C07189=1028.649,297.981,-127.130,170.913,46.438,158.974
C07190=1028.655,298.229,-127.163,170.917,46.437,158.975
C07191=1028.663,298.477,-127.195,170.922,46.437,158.975
C07192=1028.669,298.724,-127.228,170.927,46.436,158.976
C07193=1028.676,298.972,-127.261,170.931,46.436,158.976
C07194=1028.683,299.220,-127.293,170.935,46.436,158.976
C07195=1028.689,299.468,-127.326,170.941,46.435,158.977
C07196=1028.696,299.716,-127.359,170.945,46.435,158.977
C07197=1028.703,299.963,-127.391,170.949,46.434,158.978
C07198=1028.710,300.211,-127.424,170.954,46.434,158.978
C07199=1028.717,300.459,-127.457,170.959,46.432,158.978
C07200=1028.724,300.706,-127.490,170.963,46.432,158.979
C07201=1028.731,300.954,-127.523,170.967,46.432,158.979
C07202=1028.737,301.202,-127.556,170.972,46.431,158.980
C07203=1028.744,301.449,-127.588,170.977,46.431,158.980
C07204=1028.751,301.697,-127.621,170.981,46.430,158.981
C07205=1028.757,301.945,-127.654,170.986,46.430,158.981
C07206=1028.765,302.192,-127.687,170.991,46.429,158.981
C07207=1028.772,302.440,-127.720,170.995,46.429,158.982
C07208=1028.778,302.688,-127.753,171.000,46.428,158.982
C07209=1028.785,302.936,-127.786,171.005,46.428,158.983
C07210=1028.793,303.183,-127.819,171.010,46.428,158.983
C07211=1028.799,303.431,-127.852,171.014,46.427,158.984
C07212=1028.806,303.679,-127.885,171.019,46.427,158.984
C07213=1028.813,303.926,-127.917,171.024,46.426,158.985
C07214=1028.820,304.174,-127.951,171.028,46.426,158.985
C07215=1028.826,304.421,-127.984,171.033,46.425,158.986
C07216=1028.834,304.669,-128.017,171.038,46.425,158.986
C07217=1028.841,304.917,-128.050,171.042,46.424,158.986
C07218=1028.847,305.165,-128.083,171.047,46.424,158.987
C07219=1028.855,305.412,-128.117,171.052,46.423,158.987
C07220=1028.862,305.660,-128.149,171.056,46.424,158.988
C07221=1028.869,305.907,-128.183,171.062,46.423,158.988
C07222=1028.880,306.326,-128.238,171.069,46.422,158.989
C07223=1028.893,306.744,-128.294,171.077,46.422,158.990
C07224=1028.904,307.163,-128.350,171.086,46.421,158.991
C07225=1028.916,307.582,-128.406,171.093,46.420,158.992
C07226=1028.923,307.828,-128.439,171.099,46.420,158.992
C07227=1028.931,308.076,-128.473,171.103,46.419,158.992
C07228=1028.937,308.324,-128.506,171.107,46.419,158.993
C07229=1028.945,308.572,-128.539,171.113,46.419,158.994
C07230=1028.952,308.819,-128.572,171.117,46.418,158.994
C07231=1028.959,309.067,-128.606,171.122,46.418,158.994
C07232=1028.966,309.315,-128.640,171.127,46.418,158.995
C07233=1028.974,309.563,-128.672,171.132,46.417,158.996
C07234=1028.980,309.810,-128.706,171.137,46.417,158.996
C07235=1028.988,310.057,-128.740,171.141,46.417,158.997
C07236=1028.995,310.305,-128.773,171.147,46.416,158.997
C07237=1029.002,310.553,-128.806,171.151,46.416,158.997
C07238=1029.009,310.800,-128.839,171.157,46.416,158.998
C07239=1029.016,311.048,-128.873,171.161,46.415,158.998
C07240=1029.023,311.295,-128.907,171.167,46.415,158.999
C07241=1029.031,311.543,-128.941,171.171,46.415,159.000
C07242=1029.036,311.790,-128.975,171.176,46.415,159.000
C07243=1029.044,312.038,-129.009,171.181,46.415,159.001
C07244=1029.051,312.286,-129.043,171.185,46.415,159.001
C07245=1029.057,312.534,-129.077,171.190,46.415,159.002
C07246=1029.064,312.780,-129.110,171.196,46.415,159.002
C07247=1029.071,313.028,-129.144,171.200,46.415,159.003
C07248=1029.078,313.276,-129.179,171.206,46.414,159.004
C07249=1029.085,313.523,-129.213,171.210,46.415,159.004
C07250=1029.091,313.770,-129.247,171.215,46.414,159.005
C07251=1029.098,314.018,-129.281,171.220,46.414,159.005
C07252=1029.105,314.266,-129.315,171.225,46.414,159.006
C07253=1029.112,314.514,-129.349,171.230,46.414,159.006
C07254=1029.119,314.761,-129.384,171.235,46.414,159.007
C07255=1029.126,315.009,-129.418,171.240,46.414,159.008
C07256=1029.132,315.256,-129.452,171.245,46.414,159.008
C07257=1029.140,315.503,-129.486,171.251,46.414,159.009
C07258=1029.147,315.751,-129.520,171.255,46.414,159.009
C07259=1029.153,315.999,-129.555,171.260,46.414,159.010
C07260=1029.161,316.246,-129.588,171.265,46.414,159.010
C07261=1029.168,316.493,-129.623,171.270,46.414,159.011
C07262=1029.175,316.741,-129.657,171.275,46.414,159.012
C07263=1029.182,316.989,-129.691,171.280,46.414,159.012
C07264=1029.189,317.236,-129.726,171.286,46.414,159.013
C07265=1029.196,317.484,-129.760,171.290,46.414,159.013
C07266=1029.203,317.732,-129.794,171.296,46.414,159.014
C07267=1029.210,317.979,-129.829,171.300,46.414,159.015
C07268=1029.217,318.227,-129.863,171.306,46.414,159.015
C07269=1029.225,318.474,-129.897,171.311,46.414,159.016
C07270=1029.231,318.722,-129.932,171.316,46.414,159.016
C07271=1029.238,318.969,-129.966,171.321,46.414,159.017
C07272=1029.245,319.217,-130.001,171.326,46.414,159.018
C07273=1029.252,319.464,-130.035,171.331,46.414,159.018
C07274=1029.260,319.711,-130.069,171.337,46.414,159.019
C07275=1029.266,319.959,-130.104,171.341,46.414,159.020
C07276=1029.274,320.206,-130.139,171.347,46.414,159.020
C07277=1029.281,320.454,-130.173,171.351,46.415,159.021
C07278=1029.287,320.665,-130.202,171.356,46.415,159.021
C07279=1029.293,320.878,-130.232,171.360,46.414,159.022
C07280=1029.300,321.089,-130.262,171.365,46.415,159.022
C07281=1029.306,321.301,-130.291,171.370,46.415,159.023
C07282=1029.311,321.512,-130.321,171.374,46.415,159.024
C07283=1029.317,321.724,-130.350,171.379,46.415,159.024
C07284=1029.324,321.936,-130.381,171.383,46.415,159.025
C07285=1029.330,322.147,-130.410,171.388,46.415,159.025
C07286=1029.337,322.395,-130.445,171.392,46.415,159.026
C07287=1029.345,322.642,-130.479,171.398,46.415,159.026
C07288=1029.351,322.890,-130.514,171.403,46.416,159.027
C07289=1029.360,323.137,-130.549,171.409,46.416,159.028
C07290=1029.366,323.385,-130.584,171.414,46.416,159.028
C07291=1029.374,323.632,-130.618,171.419,46.416,159.029
C07292=1029.381,323.879,-130.652,171.424,46.416,159.030
C07293=1029.388,324.127,-130.688,171.429,46.416,159.030
C07294=1029.396,324.375,-130.722,171.435,46.417,159.031
C07295=1029.403,324.622,-130.757,171.441,46.417,159.032
C07296=1029.410,324.869,-130.792,171.445,46.417,159.032
C07297=1029.418,325.117,-130.827,171.451,46.417,159.033
C07298=1029.425,325.364,-130.862,171.457,46.417,159.034
C07299=1029.433,325.611,-130.896,171.461,46.417,159.034
C07300=1029.440,325.859,-130.932,171.467,46.417,159.035
C07301=1029.447,326.106,-130.966,171.473,46.418,159.036
C07302=1029.455,326.354,-131.002,171.478,46.418,159.037
C07303=1029.462,326.601,-131.036,171.483,46.418,159.037
C07304=1029.470,326.848,-131.071,171.489,46.419,159.038
C07305=1029.477,327.096,-131.106,171.494,46.419,159.039
C07306=1029.485,327.344,-131.141,171.499,46.419,159.039
C07307=1029.492,327.592,-131.177,171.505,46.419,159.040
C07308=1029.500,327.839,-131.211,171.510,46.420,159.041
C07309=1029.506,328.086,-131.246,171.516,46.420,159.042
C07310=1029.514,328.333,-131.282,171.521,46.420,159.042
C07311=1029.521,328.581,-131.318,171.526,46.421,159.043
C07312=1029.528,328.828,-131.353,171.532,46.421,159.044
C07313=1029.535,329.076,-131.389,171.538,46.421,159.044
C07314=1029.543,329.323,-131.423,171.543,46.422,159.045
C07315=1029.550,329.571,-131.459,171.548,46.422,159.046
C07316=1029.557,329.817,-131.495,171.554,46.423,159.047
C07317=1029.565,330.066,-131.530,171.559,46.423,159.047
C07318=1029.572,330.312,-131.566,171.565,46.423,159.048
C07319=1029.578,330.560,-131.601,171.571,46.424,159.049
C07320=1029.586,330.807,-131.638,171.576,46.425,159.050
C07321=1029.594,331.054,-131.672,171.581,46.425,159.050
C07322=1029.601,331.302,-131.708,171.587,46.425,159.051
C07323=1029.608,331.549,-131.743,171.593,46.426,159.052
C07324=1029.616,331.796,-131.780,171.598,46.427,159.053
C07325=1029.623,332.045,-131.815,171.604,46.426,159.053
C07326=1029.630,332.291,-131.851,171.610,46.427,159.054
C07327=1029.638,332.539,-131.887,171.615,46.428,159.055
C07328=1029.645,332.786,-131.922,171.620,46.428,159.056
C07329=1029.653,333.033,-131.958,171.626,46.429,159.057
C07330=1029.660,333.280,-131.994,171.632,46.429,159.058
C07331=1029.667,333.528,-132.029,171.638,46.429,159.058
C07332=1029.675,333.775,-132.066,171.643,46.430,159.059
C07333=1029.682,334.022,-132.101,171.649,46.431,159.060
C07334=1029.690,334.270,-132.137,171.655,46.431,159.061
C07335=1029.697,334.518,-132.173,171.660,46.432,159.061
C07336=1029.704,334.764,-132.209,171.665,46.433,159.062
C07337=1029.712,335.012,-132.245,171.671,46.433,159.063
C07338=1029.718,335.222,-132.276,171.676,46.434,159.064
C07339=1029.724,335.431,-132.307,171.681,46.434,159.064
C07340=1029.730,335.641,-132.337,171.686,46.435,159.065
C07341=1029.737,335.849,-132.368,171.690,46.435,159.066
C07342=1029.743,336.059,-132.398,171.695,46.436,159.067
C07343=1029.749,336.269,-132.429,171.700,46.437,159.067
C07344=1029.756,336.478,-132.459,171.706,46.437,159.068
C07345=1029.762,336.687,-132.490,171.711,46.437,159.069
C07346=1029.769,336.935,-132.526,171.716,46.438,159.069
C07347=1029.776,337.182,-132.562,171.721,46.439,159.070
C07348=1029.784,337.429,-132.600,171.727,46.439,159.071
C07349=1029.791,337.676,-132.636,171.734,46.440,159.072
C07350=1029.799,337.924,-132.672,171.740,46.441,159.073
C07351=1029.807,338.171,-132.708,171.745,46.441,159.074
C07352=1029.814,338.418,-132.744,171.750,46.442,159.075
C07353=1029.821,338.665,-132.780,171.756,46.443,159.075
C07354=1029.829,338.913,-132.816,171.762,46.444,159.076
C07355=1029.837,339.160,-132.853,171.768,46.444,159.077
C07356=1029.844,339.407,-132.890,171.774,46.445,159.078
C07357=1029.851,339.654,-132.926,171.781,46.446,159.079
C07358=1029.859,339.901,-132.962,171.786,46.447,159.080
C07359=1029.867,340.148,-132.999,171.791,46.447,159.081
C07360=1029.874,340.396,-133.035,171.798,46.449,159.082
C07361=1029.881,340.643,-133.072,171.803,46.449,159.083
C07362=1029.889,340.890,-133.109,171.809,46.450,159.083
C07363=1029.897,341.138,-133.145,171.816,46.451,159.084
C07364=1029.904,341.385,-133.183,171.822,46.451,159.085
C07365=1029.912,341.632,-133.219,171.828,46.452,159.086
C07366=1029.919,341.878,-133.256,171.834,46.453,159.087
C07367=1029.926,342.126,-133.293,171.840,46.454,159.088
C07368=1029.934,342.373,-133.329,171.846,46.455,159.089
C07369=1029.941,342.621,-133.366,171.851,46.456,159.090
C07370=1029.949,342.868,-133.403,171.857,46.457,159.091
C07371=1029.957,343.114,-133.440,171.863,46.458,159.092
C07372=1029.964,343.362,-133.477,171.869,46.459,159.093
C07373=1029.972,343.609,-133.514,171.875,46.459,159.094
C07374=1029.979,343.856,-133.551,171.881,46.461,159.095
C07375=1029.987,344.104,-133.588,171.888,46.462,159.096
C07376=1029.995,344.350,-133.625,171.894,46.462,159.096
C07377=1030.002,344.598,-133.662,171.900,46.463,159.097
C07378=1030.010,344.844,-133.699,171.906,46.464,159.098
C07379=1030.017,345.092,-133.736,171.912,46.466,159.099
C07380=1030.026,345.340,-133.773,171.918,46.466,159.100
C07381=1030.033,345.587,-133.811,171.924,46.467,159.101
C07382=1030.041,345.834,-133.848,171.931,46.468,159.102
C07383=1030.048,346.081,-133.885,171.937,46.469,159.103
C07384=1030.056,346.328,-133.922,171.943,46.471,159.104
C07385=1030.063,346.575,-133.960,171.949,46.471,159.105
C07386=1030.071,346.822,-133.996,171.955,46.472,159.106
C07387=1030.079,347.069,-134.034,171.961,46.473,159.107
C07388=1030.087,347.316,-134.071,171.968,46.474,159.108
C07389=1030.094,347.563,-134.109,171.974,46.476,159.109
C07390=1030.102,347.810,-134.146,171.980,46.477,159.110
C07391=1030.110,348.057,-134.183,171.986,46.478,159.111
C07392=1030.118,348.304,-134.220,171.992,46.479,159.112
C07393=1030.125,348.552,-134.258,171.999,46.480,159.113
C07394=1030.133,348.799,-134.296,172.005,46.481,159.114
C07395=1030.141,349.046,-134.333,172.011,46.482,159.115
C07396=1030.148,349.292,-134.371,172.017,46.483,159.116
C07397=1030.156,349.540,-134.409,172.024,46.484,159.117
C07398=1030.169,349.956,-134.471,172.035,46.486,159.119
C07399=1030.181,350.371,-134.535,172.046,46.488,159.121
C07400=1030.195,350.787,-134.599,172.056,46.490,159.123
C07401=1030.208,351.203,-134.662,172.067,46.492,159.124
C07402=1030.215,351.449,-134.700,172.073,46.494,159.126
C07403=1030.223,351.697,-134.738,172.080,46.495,159.127
C07404=1030.231,351.943,-134.776,172.086,46.496,159.128
C07405=1030.239,352.191,-134.813,172.092,46.497,159.129
C07406=1030.247,352.437,-134.852,172.099,46.499,159.130
C07407=1030.254,352.685,-134.889,172.106,46.500,159.131
C07408=1030.262,352.932,-134.928,172.112,46.501,159.132
C07409=1030.271,353.178,-134.965,172.119,46.503,159.133
C07410=1030.279,353.426,-135.003,172.125,46.504,159.134
C07411=1030.286,353.672,-135.042,172.131,46.506,159.135
C07412=1030.294,353.920,-135.080,172.139,46.506,159.136
C07413=1030.301,354.167,-135.118,172.145,46.508,159.138
C07414=1030.310,354.414,-135.156,172.151,46.509,159.139
C07415=1030.318,354.660,-135.194,172.157,46.510,159.140
C07416=1030.326,354.907,-135.233,172.164,46.512,159.141
C07417=1030.333,355.154,-135.270,172.172,46.514,159.142
C07418=1030.341,355.402,-135.309,172.178,46.515,159.143
C07419=1030.349,355.648,-135.347,172.184,46.516,159.144
C07420=1030.358,355.895,-135.385,172.190,46.517,159.145
C07421=1030.365,356.142,-135.423,172.198,46.519,159.146
C07422=1030.374,356.389,-135.462,172.204,46.521,159.148
C07423=1030.381,356.635,-135.500,172.211,46.522,159.149
C07424=1030.389,356.883,-135.539,172.217,46.523,159.150
C07425=1030.397,357.130,-135.577,172.225,46.525,159.151
C07426=1030.405,357.376,-135.616,172.231,46.527,159.152
C07427=1030.413,357.623,-135.654,172.237,46.528,159.153
C07428=1030.421,357.870,-135.692,172.244,46.529,159.155
C07429=1030.429,358.117,-135.731,172.252,46.531,159.156
C07430=1030.437,358.364,-135.770,172.258,46.532,159.157
C07431=1030.445,358.610,-135.809,172.265,46.534,159.158
C07432=1030.453,358.858,-135.847,172.272,46.536,159.159
C07433=1030.461,359.105,-135.886,172.278,46.537,159.160
C07434=1030.469,359.352,-135.924,172.285,46.538,159.162
C07435=1030.477,359.598,-135.963,172.292,46.540,159.163
C07436=1030.485,359.845,-136.002,172.299,46.542,159.164
C07437=1030.493,360.092,-136.041,172.305,46.543,159.165
C07438=1030.502,360.339,-136.080,172.313,46.545,159.167
C07439=1030.509,360.586,-136.119,172.319,46.546,159.168
C07440=1030.517,360.832,-136.158,172.326,46.548,159.169
C07441=1030.525,361.080,-136.197,172.333,46.549,159.170
C07442=1030.534,361.326,-136.236,172.340,46.552,159.172
C07443=1030.542,361.573,-136.275,172.347,46.553,159.173
C07444=1030.549,361.820,-136.314,172.354,46.555,159.174
C07445=1030.557,362.067,-136.353,172.361,46.557,159.175
C07446=1030.566,362.313,-136.392,172.369,46.559,159.177
C07447=1030.573,362.560,-136.432,172.375,46.560,159.178
C07448=1030.582,362.807,-136.471,172.382,46.562,159.179
C07449=1030.590,363.054,-136.510,172.389,46.563,159.180
C07450=1030.598,363.300,-136.549,172.396,46.566,159.182
C07451=1030.606,363.547,-136.589,172.404,46.567,159.183
C07452=1030.614,363.794,-136.627,172.410,46.569,159.184
C07453=1030.622,364.041,-136.667,172.418,46.571,159.186
C07454=1030.629,364.252,-136.701,172.423,46.572,159.187
C07455=1030.637,364.463,-136.735,172.430,46.574,159.188
C07456=1030.643,364.673,-136.768,172.436,46.575,159.189
C07457=1030.650,364.884,-136.802,172.441,46.577,159.190
C07458=1030.657,365.096,-136.836,172.448,46.578,159.191
C07459=1030.665,365.307,-136.869,172.454,46.580,159.192
C07460=1030.671,365.518,-136.903,172.460,46.582,159.194
C07461=1030.678,365.729,-136.937,172.466,46.583,159.195
C07462=1030.686,365.976,-136.976,172.474,46.585,159.196
C07463=1030.694,366.222,-137.016,172.480,46.587,159.197
C07464=1030.703,366.468,-137.056,172.488,46.589,159.199
C07465=1030.711,366.715,-137.096,172.495,46.591,159.200
C07466=1030.719,366.962,-137.135,172.503,46.592,159.201
C07467=1030.728,367.209,-137.175,172.509,46.595,159.203
C07468=1030.736,367.456,-137.215,172.517,46.597,159.204
C07469=1030.745,367.703,-137.254,172.525,46.598,159.205
C07470=1030.753,367.949,-137.293,172.532,46.600,159.207
C07471=1030.761,368.195,-137.334,172.539,46.602,159.208
C07472=1030.770,368.442,-137.373,172.546,46.605,159.210
C07473=1030.779,368.689,-137.413,172.554,46.606,159.211
C07474=1030.787,368.936,-137.454,172.562,46.608,159.212
C07475=1030.795,369.182,-137.493,172.569,46.610,159.214
C07476=1030.803,369.429,-137.533,172.576,46.612,159.215
C07477=1030.812,369.675,-137.573,172.583,46.615,159.217
C07478=1030.820,369.923,-137.613,172.591,46.617,159.218
C07479=1030.828,370.169,-137.654,172.599,46.619,159.219
C07480=1030.837,370.415,-137.694,172.606,46.621,159.221
C07481=1030.844,370.662,-137.734,172.613,46.623,159.222
C07482=1030.853,370.909,-137.775,172.621,46.625,159.224
C07483=1030.862,371.155,-137.815,172.628,46.627,159.225
C07484=1030.870,371.402,-137.855,172.636,46.629,159.227
C07485=1030.878,371.649,-137.896,172.644,46.632,159.228
C07486=1030.887,371.895,-137.936,172.651,46.634,159.230
C07487=1030.895,372.142,-137.976,172.659,46.636,159.231
C07488=1030.903,372.389,-138.017,172.667,46.638,159.232
C07489=1030.912,372.635,-138.057,172.674,46.640,159.234
C07490=1030.920,372.881,-138.097,172.682,46.643,159.235
C07491=1030.929,373.128,-138.138,172.689,46.645,159.237
C07492=1030.937,373.374,-138.178,172.697,46.646,159.238
C07493=1030.946,373.621,-138.219,172.705,46.649,159.240
C07494=1030.954,373.867,-138.260,172.712,46.651,159.241
C07495=1030.963,374.113,-138.300,172.720,46.653,159.243
C07496=1030.972,374.360,-138.341,172.728,46.656,159.244
C07497=1030.980,374.606,-138.382,172.736,46.658,159.246
C07498=1030.989,374.853,-138.422,172.743,46.661,159.248
C07499=1030.997,375.099,-138.463,172.751,46.663,159.249
C07500=1031.006,375.346,-138.504,172.759,46.665,159.251
C07501=1031.015,375.593,-138.544,172.767,46.667,159.252
C07502=1031.023,375.839,-138.585,172.775,46.670,159.254
C07503=1031.032,376.086,-138.627,172.783,46.672,159.255
C07504=1031.041,376.332,-138.667,172.791,46.674,159.257
C07505=1031.049,376.578,-138.708,172.798,46.677,159.258
C07506=1031.058,376.825,-138.749,172.806,46.679,159.260
C07507=1031.067,377.071,-138.789,172.814,46.681,159.261
C07508=1031.076,377.318,-138.830,172.822,46.684,159.263
C07509=1031.085,377.564,-138.872,172.830,46.686,159.265
C07510=1031.093,377.810,-138.913,172.838,46.688,159.266
C07511=1031.102,378.057,-138.954,172.846,46.691,159.268
C07512=1031.110,378.304,-138.995,172.855,46.694,159.269
C07513=1031.118,378.549,-139.037,172.863,46.696,159.271
C07514=1031.127,378.771,-139.074,172.870,46.698,159.272
C07515=1031.135,378.992,-139.111,172.877,46.701,159.274
C07516=1031.142,379.214,-139.148,172.885,46.703,159.276
C07517=1031.150,379.436,-139.185,172.891,46.705,159.277
C07518=1031.158,379.657,-139.222,172.899,46.708,159.279
C07519=1031.165,379.879,-139.260,172.906,46.710,159.280
C07520=1031.173,380.100,-139.297,172.913,46.712,159.281
C07521=1031.181,380.322,-139.334,172.921,46.715,159.283
C07522=1031.190,380.568,-139.376,172.930,46.717,159.285
C07523=1031.199,380.814,-139.417,172.938,46.720,159.286
C07524=1031.207,381.060,-139.459,172.946,46.722,159.288
C07525=1031.216,381.307,-139.501,172.954,46.725,159.290
C07526=1031.225,381.553,-139.543,172.962,46.728,159.291
C07527=1031.234,381.799,-139.585,172.971,46.730,159.293
C07528=1031.242,382.046,-139.626,172.979,46.733,159.295
C07529=1031.251,382.292,-139.668,172.987,46.736,159.297
C07530=1031.260,382.539,-139.710,172.995,46.739,159.298
C07531=1031.269,382.785,-139.751,173.004,46.741,159.300
C07532=1031.278,383.031,-139.793,173.012,46.744,159.302
C07533=1031.287,383.277,-139.836,173.020,46.747,159.303
C07534=1031.296,383.523,-139.877,173.030,46.750,159.305
C07535=1031.305,383.770,-139.919,173.038,46.752,159.307
C07536=1031.314,384.016,-139.961,173.046,46.755,159.309
C07537=1031.323,384.262,-140.003,173.054,46.758,159.310
C07538=1031.332,384.508,-140.045,173.063,46.761,159.312
C07539=1031.341,384.755,-140.087,173.072,46.764,159.314
C07540=1031.351,385.000,-140.129,173.080,46.766,159.316
C07541=1031.360,385.247,-140.171,173.089,46.769,159.318
C07542=1031.369,385.493,-140.214,173.097,46.772,159.319
C07543=1031.378,385.740,-140.255,173.106,46.775,159.321
C07544=1031.387,385.986,-140.297,173.115,46.778,159.323
C07545=1031.396,386.232,-140.339,173.124,46.781,159.325
C07546=1031.406,386.477,-140.382,173.132,46.784,159.327
C07547=1031.415,386.725,-140.425,173.141,46.786,159.328
C07548=1031.424,386.970,-140.467,173.150,46.789,159.330
C07549=1031.433,387.217,-140.509,173.158,46.792,159.332
C07550=1031.442,387.463,-140.551,173.167,46.795,159.334
C07551=1031.451,387.709,-140.595,173.176,46.798,159.336
C07552=1031.460,387.955,-140.637,173.184,46.801,159.338
C07553=1031.470,388.201,-140.679,173.193,46.804,159.339
C07554=1031.479,388.448,-140.723,173.203,46.807,159.341
C07555=1031.488,388.693,-140.765,173.211,46.810,159.343
C07556=1031.497,388.939,-140.808,173.220,46.814,159.345
C07557=1031.507,389.186,-140.850,173.229,46.816,159.347
C07558=1031.515,389.432,-140.893,173.238,46.819,159.349
C07559=1031.525,389.677,-140.936,173.247,46.823,159.351
C07560=1031.535,389.924,-140.979,173.256,46.826,159.353
C07561=1031.543,390.170,-141.022,173.265,46.829,159.355
C07562=1031.553,390.416,-141.065,173.274,46.832,159.357
C07563=1031.561,390.662,-141.108,173.283,46.835,159.359
C07564=1031.571,390.908,-141.151,173.292,46.838,159.360
C07565=1031.580,391.154,-141.194,173.301,46.842,159.363
C07566=1031.589,391.400,-141.237,173.310,46.844,159.364
C07567=1031.599,391.646,-141.281,173.319,46.848,159.366
C07568=1031.608,391.892,-141.323,173.329,46.851,159.369
C07569=1031.617,392.139,-141.366,173.337,46.854,159.370
C07570=1031.627,392.384,-141.410,173.347,46.858,159.372
C07571=1031.636,392.630,-141.453,173.356,46.861,159.375
C07572=1031.646,392.876,-141.496,173.366,46.864,159.376
C07573=1031.655,393.122,-141.540,173.374,46.868,159.378
C07574=1031.665,393.362,-141.582,173.384,46.870,159.380
C07575=1031.674,393.601,-141.624,173.393,46.874,159.382
C07576=1031.682,393.840,-141.666,173.402,46.877,159.384
C07577=1031.691,394.079,-141.708,173.411,46.880,159.386
C07578=1031.701,394.318,-141.752,173.421,46.884,159.388
C07579=1031.710,394.557,-141.794,173.429,46.887,159.390
C07580=1031.719,394.796,-141.836,173.438,46.890,159.392
C07581=1031.728,395.035,-141.879,173.448,46.894,159.394
C07582=1031.738,395.281,-141.922,173.458,46.897,159.397
C07583=1031.748,395.527,-141.966,173.466,46.901,159.399
C07584=1031.757,395.773,-142.010,173.476,46.904,159.401
C07585=1031.767,396.019,-142.054,173.486,46.908,159.403
C07586=1031.776,396.264,-142.098,173.495,46.911,159.405
C07587=1031.785,396.511,-142.142,173.505,46.915,159.407
C07588=1031.796,396.756,-142.185,173.515,46.918,159.409
C07589=1031.805,397.003,-142.229,173.525,46.922,159.411
C07590=1031.815,397.248,-142.274,173.534,46.926,159.414
C07591=1031.825,397.494,-142.318,173.543,46.929,159.416
C07592=1031.834,397.740,-142.362,173.554,46.933,159.418
C07593=1031.844,397.986,-142.406,173.563,46.936,159.420
C07594=1031.853,398.232,-142.451,173.573,46.940,159.422
C07595=1031.864,398.477,-142.494,173.583,46.943,159.424
C07596=1031.873,398.724,-142.538,173.592,46.947,159.427
C07597=1031.883,398.969,-142.583,173.602,46.951,159.429
C07598=1031.893,399.215,-142.627,173.612,46.954,159.431
C07599=1031.903,399.460,-142.671,173.622,46.958,159.433
C07600=1031.912,399.707,-142.716,173.632,46.962,159.435
C07601=1031.922,399.952,-142.760,173.642,46.965,159.438
C07602=1031.931,400.198,-142.805,173.653,46.969,159.440
C07603=1031.941,400.444,-142.849,173.663,46.973,159.442
C07604=1031.951,400.689,-142.894,173.672,46.976,159.444
C07605=1031.962,400.935,-142.939,173.683,46.980,159.447
C07606=1031.971,401.181,-142.984,173.693,46.984,159.449
C07607=1031.981,401.426,-143.028,173.703,46.988,159.451
C07608=1031.991,401.672,-143.073,173.713,46.992,159.454
C07609=1032.000,401.918,-143.117,173.723,46.996,159.456
C07610=1032.010,402.164,-143.162,173.733,46.999,159.458
C07611=1032.020,402.410,-143.207,173.744,47.004,159.461
C07612=1032.030,402.655,-143.252,173.754,47.008,159.463
C07613=1032.041,402.901,-143.298,173.764,47.012,159.465
C07614=1032.050,403.146,-143.343,173.774,47.015,159.468
C07615=1032.060,403.392,-143.388,173.785,47.020,159.470
C07616=1032.070,403.638,-143.433,173.795,47.024,159.472
C07617=1032.080,403.883,-143.479,173.805,47.027,159.475
C07618=1032.089,404.129,-143.524,173.815,47.032,159.477
C07619=1032.100,404.375,-143.569,173.826,47.035,159.480
C07620=1032.110,404.620,-143.615,173.837,47.040,159.482
C07621=1032.120,404.866,-143.660,173.847,47.043,159.484
C07622=1032.130,405.111,-143.705,173.858,47.048,159.487
C07623=1032.140,405.357,-143.750,173.868,47.052,159.489
C07624=1032.150,405.603,-143.795,173.879,47.056,159.492
C07625=1032.160,405.848,-143.842,173.890,47.060,159.494
C07626=1032.170,406.093,-143.887,173.900,47.064,159.497
C07627=1032.180,406.340,-143.933,173.910,47.068,159.499
C07628=1032.191,406.585,-143.978,173.922,47.072,159.502
C07629=1032.201,406.830,-144.024,173.932,47.077,159.504
C07630=1032.211,407.076,-144.069,173.943,47.081,159.507
C07631=1032.222,407.322,-144.115,173.954,47.085,159.509
C07632=1032.232,407.567,-144.161,173.965,47.089,159.512
C07633=1032.242,407.813,-144.207,173.976,47.094,159.514
C07634=1032.252,408.064,-144.254,173.987,47.098,159.517
C07635=1032.263,408.314,-144.301,173.998,47.103,159.520
C07636=1032.274,408.566,-144.347,174.009,47.107,159.522
C07637=1032.284,408.817,-144.394,174.020,47.111,159.525
C07638=1032.295,409.063,-144.440,174.031,47.116,159.527
C07639=1032.306,409.308,-144.486,174.043,47.120,159.530
C07640=1032.317,409.553,-144.533,174.053,47.124,159.533
C07641=1032.327,409.798,-144.578,174.065,47.129,159.535
C07642=1032.338,410.044,-144.625,174.076,47.133,159.538
C07643=1032.348,410.290,-144.671,174.087,47.137,159.540
C07644=1032.358,410.536,-144.717,174.099,47.142,159.543
C07645=1032.369,410.781,-144.764,174.109,47.146,159.546
C07646=1032.379,411.027,-144.810,174.121,47.151,159.548
C07647=1032.390,411.272,-144.857,174.132,47.156,159.551
C07648=1032.401,411.517,-144.903,174.143,47.160,159.554
C07649=1032.411,411.762,-144.950,174.155,47.164,159.557
C07650=1032.421,412.008,-144.996,174.166,47.169,159.559
C07651=1032.432,412.253,-145.043,174.178,47.174,159.562
C07652=1032.443,412.498,-145.090,174.190,47.178,159.565
C07653=1032.453,412.744,-145.137,174.200,47.183,159.567
C07654=1032.464,412.990,-145.183,174.212,47.188,159.570
C07655=1032.474,413.235,-145.230,174.224,47.192,159.573
C07656=1032.485,413.480,-145.277,174.236,47.197,159.576
C07657=1032.495,413.725,-145.324,174.248,47.201,159.579
C07658=1032.506,413.970,-145.371,174.258,47.206,159.581
C07659=1032.517,414.216,-145.418,174.270,47.211,159.584
C07660=1032.528,414.461,-145.465,174.282,47.215,159.587
C07661=1032.538,414.707,-145.512,174.294,47.220,159.590
C07662=1032.550,414.952,-145.559,174.306,47.225,159.593
C07663=1032.560,415.198,-145.606,174.318,47.229,159.595
C07664=1032.572,415.443,-145.654,174.330,47.234,159.598
C07665=1032.582,415.688,-145.701,174.342,47.239,159.601
C07666=1032.593,415.934,-145.748,174.354,47.244,159.604
C07667=1032.604,416.179,-145.795,174.366,47.249,159.607
C07668=1032.615,416.424,-145.843,174.378,47.254,159.610
C07669=1032.626,416.669,-145.890,174.390,47.259,159.613
C07670=1032.637,416.917,-145.938,174.402,47.264,159.616
C07671=1032.649,417.165,-145.987,174.414,47.268,159.619
C07672=1032.659,417.413,-146.035,174.426,47.273,159.622
C07673=1032.671,417.660,-146.083,174.439,47.279,159.625
C07674=1032.681,417.905,-146.130,174.451,47.284,159.628
C07675=1032.692,418.151,-146.179,174.464,47.289,159.631
C07676=1032.703,418.396,-146.227,174.476,47.294,159.634
C07677=1032.715,418.640,-146.274,174.489,47.299,159.637
C07678=1032.726,418.886,-146.323,174.501,47.304,159.640
C07679=1032.737,419.131,-146.371,174.513,47.309,159.643
C07680=1032.748,419.377,-146.419,174.526,47.314,159.646
C07681=1032.759,419.621,-146.467,174.539,47.319,159.649
C07682=1032.770,419.866,-146.515,174.551,47.324,159.652
C07683=1032.781,420.112,-146.563,174.563,47.329,159.655
C07684=1032.792,420.357,-146.611,174.576,47.335,159.658
C07685=1032.804,420.602,-146.659,174.589,47.340,159.661
C07686=1032.815,420.847,-146.707,174.602,47.345,159.665
C07687=1032.827,421.092,-146.756,174.614,47.350,159.668
C07688=1032.838,421.338,-146.805,174.627,47.356,159.671
C07689=1032.850,421.582,-146.853,174.640,47.361,159.674
C07690=1032.861,421.827,-146.901,174.653,47.366,159.677
C07691=1032.872,422.073,-146.950,174.666,47.371,159.680
C07692=1032.884,422.317,-146.999,174.679,47.377,159.683
C07693=1032.895,422.563,-147.047,174.692,47.382,159.687
C07694=1032.907,422.826,-147.099,174.706,47.388,159.690
C07695=1032.920,423.089,-147.152,174.720,47.394,159.694
C07696=1032.932,423.353,-147.204,174.735,47.399,159.697
C07697=1032.945,423.616,-147.258,174.749,47.405,159.701
C07698=1032.956,423.861,-147.307,174.761,47.411,159.704
C07699=1032.967,424.106,-147.355,174.775,47.416,159.707
C07700=1032.979,424.351,-147.404,174.789,47.422,159.711
C07701=1032.990,424.595,-147.454,174.802,47.427,159.714
C07702=1033.002,424.841,-147.503,174.815,47.433,159.717
C07703=1033.014,425.085,-147.552,174.829,47.438,159.721
C07704=1033.025,425.330,-147.601,174.843,47.444,159.724
C07705=1033.038,425.575,-147.650,174.856,47.449,159.727
C07706=1033.049,425.820,-147.699,174.870,47.455,159.731
C07707=1033.062,426.065,-147.749,174.883,47.461,159.734
C07708=1033.073,426.310,-147.798,174.896,47.466,159.738
C07709=1033.085,426.554,-147.848,174.910,47.472,159.741
C07710=1033.096,426.800,-147.898,174.924,47.478,159.745
C07711=1033.108,427.045,-147.947,174.938,47.484,159.748
C07712=1033.120,427.289,-147.997,174.952,47.489,159.752
C07713=1033.132,427.534,-148.047,174.966,47.495,159.755
C07714=1033.143,427.779,-148.096,174.980,47.501,159.758
C07715=1033.156,428.023,-148.146,174.994,47.507,159.762
C07716=1033.167,428.269,-148.197,175.008,47.513,159.766
C07717=1033.179,428.513,-148.247,175.022,47.518,159.769
C07718=1033.191,428.758,-148.297,175.036,47.525,159.773
C07719=1033.204,429.002,-148.347,175.051,47.530,159.776
C07720=1033.215,429.247,-148.397,175.065,47.536,159.780
C07721=1033.227,429.492,-148.447,175.079,47.542,159.784
C07722=1033.239,429.736,-148.497,175.093,47.548,159.787
C07723=1033.251,429.981,-148.547,175.108,47.554,159.791
C07724=1033.263,430.226,-148.599,175.123,47.560,159.795
C07725=1033.275,430.470,-148.648,175.137,47.566,159.798
C07726=1033.287,430.715,-148.699,175.151,47.572,159.802
C07727=1033.300,430.959,-148.749,175.166,47.578,159.806
C07728=1033.312,431.204,-148.799,175.180,47.584,159.809
C07729=1033.324,431.448,-148.851,175.195,47.590,159.813
C07730=1033.336,431.693,-148.901,175.210,47.596,159.817
C07731=1033.349,431.937,-148.952,175.225,47.603,159.821
C07732=1033.362,432.181,-149.003,175.240,47.609,159.824
C07733=1033.373,432.427,-149.053,175.255,47.615,159.828
C07734=1033.386,432.671,-149.104,175.269,47.621,159.832
C07735=1033.399,432.916,-149.155,175.285,47.627,159.836
C07736=1033.412,433.160,-149.206,175.300,47.634,159.840
C07737=1033.424,433.404,-149.257,175.315,47.640,159.843
C07738=1033.436,433.649,-149.308,175.330,47.646,159.847
C07739=1033.449,433.894,-149.359,175.345,47.652,159.851
C07740=1033.462,434.138,-149.410,175.360,47.659,159.855
C07741=1033.474,434.382,-149.462,175.376,47.665,159.859
C07742=1033.487,434.627,-149.513,175.391,47.671,159.863
C07743=1033.499,434.872,-149.564,175.407,47.678,159.867
C07744=1033.512,435.115,-149.616,175.422,47.684,159.871
C07745=1033.525,435.360,-149.667,175.438,47.690,159.875
C07746=1033.537,435.604,-149.719,175.453,47.697,159.879
C07747=1033.551,435.849,-149.770,175.469,47.704,159.883
C07748=1033.563,436.093,-149.822,175.484,47.710,159.887
C07749=1033.576,436.337,-149.874,175.500,47.717,159.891
C07750=1033.588,436.582,-149.926,175.516,47.723,159.895
C07751=1033.602,436.826,-149.978,175.533,47.730,159.899
C07752=1033.614,437.070,-150.030,175.548,47.736,159.903
C07753=1033.627,437.314,-150.082,175.564,47.743,159.908
C07754=1033.641,437.569,-150.136,175.581,47.750,159.912
C07755=1033.654,437.824,-150.190,175.598,47.757,159.916
C07756=1033.668,438.080,-150.245,175.615,47.764,159.921
C07757=1033.682,438.335,-150.300,175.631,47.771,159.925
C07758=1033.694,438.580,-150.352,175.648,47.778,159.929
C07759=1033.708,438.824,-150.404,175.664,47.784,159.934
C07760=1033.720,439.067,-150.457,175.680,47.791,159.938
C07761=1033.734,439.311,-150.509,175.697,47.798,159.942
C07762=1033.747,439.555,-150.562,175.714,47.805,159.946
C07763=1033.760,439.800,-150.614,175.731,47.811,159.951
C07764=1033.774,440.044,-150.667,175.747,47.819,159.955
C07765=1033.786,440.288,-150.720,175.764,47.825,159.959
C07766=1033.800,440.532,-150.773,175.780,47.832,159.964
C07767=1033.813,440.776,-150.825,175.798,47.839,159.968
C07768=1033.826,441.020,-150.879,175.815,47.846,159.973
C07769=1033.840,441.264,-150.932,175.831,47.854,159.977
C07770=1033.853,441.507,-150.984,175.849,47.861,159.982
C07771=1033.867,441.752,-151.038,175.866,47.867,159.986
C07772=1033.880,441.996,-151.091,175.882,47.875,159.991
C07773=1033.894,442.240,-151.144,175.900,47.882,159.995
C07774=1033.907,442.484,-151.197,175.917,47.888,159.999
C07775=1033.921,442.728,-151.250,175.935,47.896,160.004
C07776=1033.935,442.971,-151.304,175.952,47.903,160.009
C07777=1033.948,443.215,-151.357,175.969,47.910,160.013
C07778=1033.962,443.458,-151.410,175.987,47.917,160.018
C07779=1033.976,443.701,-151.464,176.005,47.924,160.023
C07780=1033.990,443.944,-151.517,176.022,47.931,160.027
C07781=1034.004,444.188,-151.570,176.040,47.939,160.032
C07782=1034.020,444.431,-151.621,176.057,47.946,160.036
C07783=1034.036,444.675,-151.673,176.076,47.952,160.041
C07784=1034.051,444.919,-151.725,176.093,47.959,160.045
C07785=1034.068,445.162,-151.776,176.112,47.966,160.050
C07786=1034.085,445.406,-151.826,176.130,47.972,160.054
C07787=1034.103,445.650,-151.877,176.148,47.979,160.059
C07788=1034.122,445.894,-151.926,176.167,47.985,160.063
C07789=1034.140,446.138,-151.976,176.185,47.992,160.068
C07790=1034.160,446.382,-152.024,176.203,47.998,160.073
C07791=1034.179,446.626,-152.073,176.222,48.004,160.077
C07792=1034.200,446.870,-152.120,176.240,48.011,160.082
C07793=1034.221,447.115,-152.168,176.259,48.016,160.086
C07794=1034.242,447.359,-152.215,176.278,48.022,160.091
C07795=1034.263,447.603,-152.262,176.297,48.029,160.095
C07796=1034.285,447.848,-152.308,176.316,48.034,160.099
C07797=1034.309,448.092,-152.354,176.335,48.040,160.104
C07798=1034.333,448.337,-152.399,176.354,48.046,160.108
C07799=1034.356,448.582,-152.445,176.373,48.051,160.113
C07800=1034.381,448.827,-152.488,176.392,48.057,160.117
C07801=1034.405,449.072,-152.533,176.412,48.062,160.122
C07802=1034.431,449.318,-152.577,176.431,48.068,160.126
C07803=1034.457,449.563,-152.620,176.451,48.073,160.130
C07804=1034.484,449.808,-152.662,176.471,48.078,160.135
C07805=1034.511,450.053,-152.705,176.490,48.083,160.139
C07806=1034.538,450.298,-152.747,176.510,48.088,160.143
C07807=1034.567,450.543,-152.788,176.530,48.093,160.148
C07808=1034.595,450.789,-152.829,176.550,48.098,160.152
C07809=1034.624,451.034,-152.870,176.570,48.103,160.157
C07810=1034.653,451.280,-152.910,176.591,48.107,160.161
C07811=1034.685,451.525,-152.950,176.611,48.112,160.165
C07812=1034.714,451.771,-152.989,176.631,48.117,160.170
C07813=1034.746,452.016,-153.028,176.651,48.121,160.174
C07814=1034.798,452.413,-153.090,176.685,48.129,160.181
C07815=1034.851,452.809,-153.151,176.718,48.136,160.188
C07816=1034.564,452.870,-153.479,176.721,48.203,160.209
C07817=1034.514,452.499,-153.422,176.690,48.197,160.203
C07818=1034.465,452.126,-153.364,176.659,48.191,160.196
C07819=1034.434,451.881,-153.326,176.638,48.186,160.192
C07820=1034.403,451.636,-153.286,176.618,48.182,160.188
C07821=1034.373,451.390,-153.247,176.598,48.177,160.183
C07822=1034.343,451.144,-153.206,176.577,48.172,160.179
C07823=1034.313,450.899,-153.166,176.557,48.168,160.175
C07824=1034.284,450.654,-153.125,176.537,48.163,160.170
C07825=1034.256,450.408,-153.084,176.517,48.158,160.166
C07826=1034.228,450.163,-153.042,176.497,48.153,160.162
C07827=1034.201,449.917,-153.000,176.477,48.148,160.157
C07828=1034.174,449.672,-152.958,176.457,48.143,160.153
C07829=1034.147,449.427,-152.915,176.437,48.138,160.148
C07830=1034.122,449.182,-152.871,176.418,48.132,160.144
C07831=1034.096,448.938,-152.828,176.398,48.127,160.140
C07832=1034.072,448.692,-152.783,176.379,48.122,160.135
C07833=1034.048,448.447,-152.738,176.360,48.117,160.131
C07834=1034.024,448.203,-152.694,176.341,48.111,160.126
C07835=1034.001,447.958,-152.647,176.322,48.105,160.122
C07836=1033.978,447.714,-152.602,176.303,48.100,160.118
C07837=1033.955,447.469,-152.555,176.283,48.094,160.113
C07838=1033.934,447.224,-152.508,176.264,48.088,160.109
C07839=1033.913,446.979,-152.461,176.245,48.082,160.104
C07840=1033.893,446.736,-152.414,176.227,48.076,160.100
C07841=1033.872,446.491,-152.365,176.209,48.070,160.095
C07842=1033.853,446.247,-152.317,176.189,48.064,160.091
C07843=1033.834,446.004,-152.268,176.171,48.058,160.086
C07844=1033.815,445.759,-152.218,176.153,48.052,160.082
C07845=1033.797,445.515,-152.169,176.134,48.045,160.077
C07846=1033.779,445.272,-152.118,176.116,48.039,160.073
C07847=1033.762,445.027,-152.067,176.098,48.032,160.068
C07848=1033.746,444.784,-152.016,176.080,48.026,160.064
C07849=1033.730,444.541,-151.965,176.062,48.019,160.059
C07850=1033.715,444.297,-151.913,176.044,48.012,160.054
C07851=1033.700,444.054,-151.861,176.027,48.005,160.050
C07852=1033.685,443.810,-151.807,176.008,47.998,160.045
C07853=1033.672,443.568,-151.754,175.991,47.991,160.040
C07854=1033.658,443.325,-151.701,175.973,47.984,160.036
C07855=1033.644,443.081,-151.648,175.956,47.977,160.031
C07856=1033.630,442.837,-151.594,175.938,47.970,160.027
C07857=1033.617,442.593,-151.541,175.920,47.963,160.022
C07858=1033.603,442.349,-151.488,175.903,47.956,160.018
C07859=1033.589,442.105,-151.435,175.886,47.949,160.013
C07860=1033.576,441.861,-151.382,175.869,47.942,160.009
C07861=1033.562,441.618,-151.328,175.852,47.935,160.004
C07862=1033.549,441.374,-151.275,175.834,47.928,160.000
C07863=1033.536,441.129,-151.223,175.817,47.921,159.995
C07864=1033.522,440.886,-151.170,175.801,47.914,159.991
C07865=1033.508,440.641,-151.116,175.784,47.907,159.986
C07866=1033.495,440.397,-151.064,175.766,47.900,159.982
C07867=1033.481,440.153,-151.011,175.750,47.893,159.978
C07868=1033.469,439.909,-150.958,175.733,47.887,159.973
C07869=1033.455,439.666,-150.906,175.717,47.880,159.969
C07870=1033.443,439.421,-150.853,175.700,47.873,159.965
C07871=1033.430,439.177,-150.800,175.683,47.866,159.960
C07872=1033.416,438.933,-150.748,175.666,47.860,159.956
C07873=1033.403,438.689,-150.695,175.650,47.853,159.952
C07874=1033.389,438.445,-150.643,175.633,47.846,159.948
C07875=1033.376,438.188,-150.588,175.617,47.839,159.943
C07876=1033.363,437.932,-150.534,175.600,47.832,159.939
C07877=1033.348,437.676,-150.479,175.583,47.826,159.934
C07878=1033.336,437.420,-150.424,175.565,47.819,159.930
C07879=1033.322,437.175,-150.372,175.550,47.812,159.926
C07880=1033.309,436.931,-150.320,175.534,47.805,159.922
C07881=1033.296,436.687,-150.268,175.518,47.799,159.918
C07882=1033.284,436.443,-150.216,175.502,47.792,159.914
C07883=1033.271,436.198,-150.165,175.486,47.786,159.910
C07884=1033.258,435.954,-150.113,175.470,47.780,159.905
C07885=1033.245,435.710,-150.061,175.454,47.773,159.901
C07886=1033.233,435.465,-150.009,175.438,47.767,159.897
C07887=1033.220,435.222,-149.958,175.424,47.760,159.893
C07888=1033.207,434.977,-149.907,175.408,47.754,159.889
C07889=1033.195,434.732,-149.855,175.392,47.748,159.885
C07890=1033.181,434.488,-149.803,175.377,47.741,159.881
C07891=1033.169,434.243,-149.752,175.361,47.735,159.877
C07892=1033.157,433.999,-149.701,175.346,47.729,159.874
C07893=1033.143,433.754,-149.650,175.330,47.723,159.870
C07894=1033.132,433.510,-149.599,175.315,47.716,159.866
C07895=1033.119,433.266,-149.548,175.300,47.710,159.862
C07896=1033.106,433.021,-149.497,175.285,47.704,159.858
C07897=1033.093,432.776,-149.446,175.270,47.698,159.854
C07898=1033.081,432.532,-149.394,175.255,47.692,159.850
C07899=1033.069,432.287,-149.344,175.240,47.686,159.847
C07900=1033.056,432.043,-149.293,175.225,47.679,159.843
C07901=1033.044,431.799,-149.243,175.210,47.674,159.839
C07902=1033.031,431.554,-149.192,175.196,47.667,159.835
C07903=1033.019,431.309,-149.141,175.180,47.662,159.832
C07904=1033.007,431.065,-149.091,175.166,47.655,159.828
C07905=1032.995,430.820,-149.040,175.151,47.650,159.824
C07906=1032.982,430.575,-148.990,175.136,47.643,159.820
C07907=1032.970,430.331,-148.940,175.122,47.638,159.817
C07908=1032.958,430.086,-148.889,175.107,47.632,159.813
C07909=1032.946,429.842,-148.839,175.093,47.626,159.809
C07910=1032.934,429.597,-148.789,175.078,47.620,159.806
C07911=1032.922,429.352,-148.739,175.064,47.614,159.802
C07912=1032.910,429.107,-148.688,175.050,47.608,159.799
C07913=1032.898,428.862,-148.638,175.036,47.602,159.795
C07914=1032.886,428.618,-148.588,175.021,47.597,159.791
C07915=1032.874,428.373,-148.538,175.007,47.591,159.788
C07916=1032.861,428.129,-148.488,174.993,47.585,159.784
C07917=1032.851,427.884,-148.438,174.979,47.579,159.781
C07918=1032.838,427.639,-148.388,174.965,47.574,159.777
C07919=1032.826,427.395,-148.338,174.951,47.568,159.774
C07920=1032.814,427.150,-148.288,174.937,47.562,159.770
C07921=1032.803,426.906,-148.239,174.923,47.556,159.767
C07922=1032.791,426.660,-148.189,174.909,47.551,159.763
C07923=1032.778,426.415,-148.139,174.895,47.546,159.760
C07924=1032.767,426.171,-148.090,174.882,47.540,159.756
C07925=1032.755,425.927,-148.040,174.868,47.534,159.753
C07926=1032.743,425.681,-147.991,174.854,47.529,159.750
C07927=1032.732,425.436,-147.942,174.840,47.523,159.746
C07928=1032.720,425.191,-147.893,174.827,47.518,159.743
C07929=1032.709,424.946,-147.844,174.814,47.512,159.739
C07930=1032.697,424.702,-147.794,174.800,47.507,159.736
C07931=1032.685,424.457,-147.745,174.786,47.501,159.733
C07932=1032.673,424.212,-147.696,174.773,47.496,159.729
C07933=1032.662,423.967,-147.647,174.759,47.491,159.726
C07934=1032.651,423.722,-147.598,174.747,47.485,159.723
C07935=1032.638,423.457,-147.545,174.731,47.479,159.719
C07936=1032.626,423.191,-147.491,174.718,47.473,159.716
C07937=1032.614,422.925,-147.438,174.704,47.467,159.712
C07938=1032.601,422.660,-147.386,174.689,47.462,159.709
C07939=1032.589,422.413,-147.337,174.676,47.456,159.705
C07940=1032.577,422.169,-147.288,174.663,47.451,159.702
C07941=1032.566,421.924,-147.240,174.650,47.447,159.699
C07942=1032.555,421.679,-147.191,174.637,47.441,159.696
C07943=1032.543,421.434,-147.143,174.623,47.436,159.693
C07944=1032.531,421.189,-147.094,174.611,47.431,159.690
C07945=1032.520,420.944,-147.046,174.598,47.425,159.686
C07946=1032.509,420.698,-146.998,174.585,47.420,159.683
C07947=1032.498,420.453,-146.950,174.573,47.415,159.680
C07948=1032.486,420.209,-146.901,174.560,47.410,159.677
C07949=1032.475,419.964,-146.853,174.547,47.405,159.674
C07950=1032.464,419.719,-146.805,174.535,47.400,159.671
C07951=1032.453,419.473,-146.757,174.522,47.395,159.668
C07952=1032.441,419.228,-146.709,174.510,47.390,159.665
C07953=1032.430,418.983,-146.661,174.497,47.385,159.662
C07954=1032.420,418.738,-146.613,174.484,47.380,159.659
C07955=1032.409,418.493,-146.564,174.472,47.374,159.656
C07956=1032.397,418.248,-146.517,174.459,47.369,159.653
C07957=1032.387,418.002,-146.469,174.448,47.365,159.650
C07958=1032.376,417.757,-146.421,174.435,47.360,159.647
C07959=1032.364,417.512,-146.373,174.422,47.355,159.644
C07960=1032.354,417.267,-146.326,174.410,47.350,159.641
C07961=1032.342,417.021,-146.278,174.398,47.345,159.638
C07962=1032.332,416.777,-146.230,174.386,47.341,159.635
C07963=1032.320,416.531,-146.183,174.374,47.335,159.632
C07964=1032.310,416.286,-146.136,174.362,47.330,159.629
C07965=1032.298,416.041,-146.088,174.350,47.326,159.626
C07966=1032.288,415.795,-146.041,174.338,47.321,159.623
C07967=1032.277,415.550,-145.994,174.326,47.316,159.620
C07968=1032.266,415.305,-145.946,174.314,47.312,159.618
C07969=1032.255,415.059,-145.899,174.302,47.307,159.615
C07970=1032.244,414.814,-145.852,174.290,47.302,159.612
C07971=1032.233,414.569,-145.805,174.278,47.298,159.609
C07972=1032.223,414.323,-145.758,174.266,47.293,159.606
C07973=1032.212,414.078,-145.711,174.254,47.289,159.603
C07974=1032.201,413.833,-145.664,174.242,47.283,159.600
C07975=1032.190,413.587,-145.617,174.230,47.279,159.598
C07976=1032.179,413.342,-145.570,174.219,47.274,159.595
C07977=1032.169,413.097,-145.523,174.208,47.270,159.592
C07978=1032.158,412.852,-145.476,174.196,47.266,159.589
C07979=1032.148,412.605,-145.429,174.184,47.261,159.587
C07980=1032.137,412.360,-145.383,174.172,47.256,159.584
C07981=1032.126,412.115,-145.336,174.162,47.252,159.581
C07982=1032.115,411.870,-145.289,174.150,47.247,159.578
C07983=1032.106,411.624,-145.242,174.138,47.243,159.576
C07984=1032.095,411.379,-145.196,174.127,47.238,159.573
C07985=1032.085,411.133,-145.149,174.116,47.234,159.570
C07986=1032.074,410.888,-145.103,174.104,47.230,159.568
C07987=1032.063,410.643,-145.057,174.093,47.225,159.565
C07988=1032.053,410.398,-145.010,174.082,47.221,159.562
C07989=1032.042,410.152,-144.964,174.070,47.217,159.560
C07990=1032.032,409.906,-144.918,174.059,47.212,159.557
C07991=1032.021,409.661,-144.872,174.048,47.208,159.554
C07992=1032.011,409.415,-144.826,174.037,47.203,159.552
C07993=1032.000,409.170,-144.780,174.026,47.199,159.549
C07994=1031.990,408.924,-144.734,174.015,47.195,159.547
C07995=1031.979,408.669,-144.685,174.004,47.191,159.544
C07996=1031.968,408.413,-144.638,173.992,47.186,159.541
C07997=1031.957,408.157,-144.590,173.980,47.182,159.539
C07998=1031.941,407.771,-144.518,173.962,47.175,159.535
C07999=1031.924,407.395,-144.448,173.946,47.169,159.531
C08000=1031.915,407.149,-144.402,173.936,47.165,159.528
C08001=1031.904,406.903,-144.356,173.924,47.160,159.526
C08002=1031.894,406.658,-144.311,173.914,47.156,159.523
C08003=1031.884,406.412,-144.265,173.903,47.153,159.521
C08004=1031.874,406.167,-144.220,173.892,47.148,159.518
C08005=1031.863,405.921,-144.174,173.882,47.144,159.516
C08006=1031.853,405.676,-144.128,173.871,47.140,159.513
C08007=1031.843,405.431,-144.083,173.860,47.136,159.511
C08008=1031.833,405.184,-144.037,173.850,47.132,159.508
C08009=1031.823,404.939,-143.992,173.839,47.128,159.506
C08010=1031.813,404.693,-143.946,173.828,47.124,159.504
C08011=1031.803,404.448,-143.902,173.818,47.120,159.501
C08012=1031.792,404.202,-143.856,173.808,47.116,159.499
C08013=1031.783,403.956,-143.811,173.797,47.112,159.496
C08014=1031.773,403.711,-143.766,173.787,47.108,159.494
C08015=1031.762,403.465,-143.720,173.776,47.105,159.492
C08016=1031.753,403.220,-143.675,173.765,47.100,159.489
C08017=1031.742,402.974,-143.630,173.755,47.096,159.487
C08018=1031.733,402.728,-143.585,173.745,47.092,159.485
C08019=1031.724,402.482,-143.540,173.735,47.089,159.482
C08020=1031.714,402.237,-143.495,173.725,47.085,159.480
C08021=1031.704,401.991,-143.450,173.715,47.081,159.478
C08022=1031.694,401.745,-143.405,173.704,47.077,159.475
C08023=1031.683,401.500,-143.361,173.694,47.073,159.473
C08024=1031.673,401.254,-143.316,173.684,47.070,159.471
C08025=1031.663,401.008,-143.271,173.674,47.066,159.468
C08026=1031.654,400.763,-143.226,173.664,47.062,159.466
C08027=1031.644,400.516,-143.182,173.654,47.058,159.464
C08028=1031.635,400.271,-143.137,173.644,47.055,159.462
C08029=1031.625,400.025,-143.092,173.634,47.051,159.459
C08030=1031.615,399.779,-143.048,173.624,47.047,159.457
C08031=1031.604,399.533,-143.003,173.614,47.044,159.455
C08032=1031.595,399.288,-142.959,173.604,47.040,159.453
C08033=1031.585,399.042,-142.915,173.593,47.036,159.450
C08034=1031.576,398.796,-142.870,173.584,47.033,159.448
C08035=1031.565,398.550,-142.826,173.573,47.029,159.446
C08036=1031.556,398.304,-142.782,173.564,47.026,159.444
C08037=1031.546,398.059,-142.737,173.554,47.022,159.442
C08038=1031.536,397.813,-142.694,173.544,47.019,159.439
C08039=1031.527,397.567,-142.650,173.534,47.015,159.437
C08040=1031.517,397.321,-142.605,173.525,47.012,159.435
C08041=1031.507,397.076,-142.562,173.515,47.008,159.433
C08042=1031.498,396.830,-142.518,173.505,47.005,159.431
C08043=1031.489,396.584,-142.473,173.495,47.001,159.429
C08044=1031.478,396.338,-142.430,173.485,46.998,159.426
C08045=1031.469,396.092,-142.386,173.477,46.994,159.424
C08046=1031.460,395.846,-142.342,173.467,46.991,159.422
C08047=1031.450,395.601,-142.299,173.457,46.988,159.420
C08048=1031.441,395.355,-142.254,173.447,46.984,159.418
C08049=1031.431,395.108,-142.210,173.438,46.981,159.416
C08050=1031.421,394.863,-142.167,173.428,46.978,159.414
C08051=1031.406,394.447,-142.093,173.412,46.971,159.410
C08052=1031.390,394.032,-142.019,173.397,46.966,159.407
C08053=1031.374,393.617,-141.946,173.380,46.961,159.403
C08054=1031.358,393.202,-141.872,173.365,46.955,159.400
C08055=1031.348,392.955,-141.829,173.355,46.952,159.398
C08056=1031.339,392.710,-141.786,173.346,46.949,159.396
C08057=1031.329,392.464,-141.742,173.337,46.945,159.394
C08058=1031.319,392.218,-141.699,173.328,46.942,159.392
C08059=1031.311,391.972,-141.656,173.318,46.939,159.390
C08060=1031.301,391.726,-141.613,173.310,46.936,159.388
C08061=1031.292,391.480,-141.570,173.300,46.933,159.386
C08062=1031.282,391.234,-141.526,173.290,46.930,159.384
C08063=1031.274,390.988,-141.483,173.282,46.926,159.382
C08064=1031.264,390.741,-141.440,173.272,46.924,159.380
C08065=1031.255,390.496,-141.397,173.263,46.920,159.378
C08066=1031.246,390.250,-141.354,173.255,46.917,159.376
C08067=1031.237,390.003,-141.311,173.245,46.914,159.374
C08068=1031.227,389.758,-141.268,173.237,46.911,159.373
C08069=1031.217,389.511,-141.226,173.227,46.908,159.370
C08070=1031.209,389.265,-141.183,173.219,46.905,159.369
C08071=1031.199,389.019,-141.140,173.209,46.902,159.367
C08072=1031.190,388.773,-141.097,173.201,46.899,159.365
C08073=1031.181,388.527,-141.054,173.191,46.896,159.363
C08074=1031.172,388.280,-141.012,173.183,46.893,159.361
C08075=1031.162,388.035,-140.969,173.174,46.890,159.359
C08076=1031.154,387.789,-140.926,173.165,46.887,159.357
C08077=1031.145,387.543,-140.884,173.156,46.884,159.355
C08078=1031.135,387.296,-140.842,173.148,46.881,159.354
C08079=1031.126,387.050,-140.799,173.138,46.878,159.352
C08080=1031.117,386.804,-140.756,173.130,46.875,159.350
C08081=1031.108,386.558,-140.714,173.121,46.873,159.348
C08082=1031.099,386.311,-140.672,173.112,46.870,159.346
C08083=1031.090,386.065,-140.630,173.104,46.867,159.344
C08084=1031.080,385.819,-140.587,173.095,46.864,159.343
C08085=1031.071,385.573,-140.546,173.086,46.862,159.341
C08086=1031.062,385.327,-140.503,173.077,46.858,159.339
C08087=1031.053,385.080,-140.461,173.069,46.856,159.337
C08088=1031.043,384.834,-140.419,173.060,46.853,159.335
C08089=1031.034,384.588,-140.377,173.051,46.850,159.334
C08090=1031.026,384.341,-140.335,173.043,46.848,159.332
C08091=1031.016,384.096,-140.293,173.035,46.845,159.330
C08092=1031.007,383.849,-140.251,173.026,46.842,159.328
C08093=1030.998,383.603,-140.210,173.017,46.840,159.327
C08094=1030.990,383.357,-140.168,173.009,46.837,159.325
C08095=1030.980,383.111,-140.125,173.001,46.834,159.323
C08096=1030.971,382.865,-140.084,172.992,46.831,159.321
C08097=1030.962,382.618,-140.042,172.984,46.829,159.320
C08098=1030.953,382.372,-140.000,172.976,46.826,159.318
C08099=1030.945,382.125,-139.959,172.967,46.824,159.316
C08100=1030.936,381.879,-139.917,172.958,46.821,159.315
C08101=1030.927,381.632,-139.874,172.950,46.818,159.313
C08102=1030.918,381.386,-139.833,172.942,46.816,159.311
C08103=1030.910,381.140,-139.791,172.934,46.813,159.310
C08104=1030.901,380.894,-139.750,172.926,46.811,159.308
C08105=1030.892,380.648,-139.708,172.917,46.808,159.306
C08106=1030.883,380.401,-139.666,172.909,46.805,159.304
C08107=1030.875,380.179,-139.630,172.901,46.803,159.303
C08108=1030.867,379.956,-139.592,172.894,46.801,159.302
C08109=1030.859,379.734,-139.554,172.886,46.799,159.300
C08110=1030.852,379.510,-139.516,172.879,46.796,159.299
C08111=1030.844,379.289,-139.479,172.872,46.794,159.297
C08112=1030.836,379.066,-139.442,172.864,46.792,159.296
C08113=1030.828,378.843,-139.404,172.857,46.789,159.294
C08114=1030.821,378.620,-139.367,172.849,46.787,159.293
C08115=1030.812,378.375,-139.326,172.841,46.785,159.291
C08116=1030.804,378.128,-139.285,172.833,46.782,159.289
C08117=1030.795,377.881,-139.243,172.825,46.780,159.288
C08118=1030.786,377.636,-139.201,172.818,46.778,159.286
C08119=1030.777,377.389,-139.161,172.810,46.775,159.285
C08120=1030.768,377.142,-139.120,172.802,46.773,159.283
C08121=1030.759,376.896,-139.078,172.794,46.771,159.282
C08122=1030.751,376.650,-139.038,172.786,46.768,159.280
C08123=1030.742,376.403,-138.997,172.778,46.766,159.278
C08124=1030.734,376.156,-138.957,172.770,46.764,159.277
C08125=1030.725,375.910,-138.915,172.762,46.762,159.275
C08126=1030.716,375.663,-138.875,172.754,46.759,159.274
C08127=1030.708,375.417,-138.834,172.746,46.757,159.272
C08128=1030.699,375.170,-138.793,172.738,46.755,159.271
C08129=1030.690,374.924,-138.753,172.730,46.753,159.269
C08130=1030.682,374.677,-138.712,172.723,46.750,159.268
C08131=1030.674,374.431,-138.671,172.715,46.748,159.266
C08132=1030.664,374.184,-138.631,172.707,46.746,159.265
C08133=1030.656,373.938,-138.590,172.699,46.743,159.263
C08134=1030.648,373.691,-138.549,172.691,46.742,159.261
C08135=1030.639,373.445,-138.509,172.683,46.740,159.260
C08136=1030.630,373.198,-138.468,172.676,46.737,159.259
C08137=1030.622,372.952,-138.427,172.668,46.735,159.257
C08138=1030.613,372.706,-138.387,172.660,46.733,159.256
C08139=1030.605,372.459,-138.346,172.653,46.731,159.254
C08140=1030.597,372.212,-138.306,172.645,46.729,159.253
C08141=1030.588,371.966,-138.266,172.638,46.727,159.251
C08142=1030.580,371.719,-138.225,172.630,46.724,159.250
C08143=1030.572,371.473,-138.185,172.622,46.722,159.248
C08144=1030.563,371.227,-138.145,172.615,46.720,159.247
C08145=1030.555,370.979,-138.105,172.607,46.718,159.245
C08146=1030.546,370.733,-138.064,172.599,46.716,159.244
C08147=1030.538,370.487,-138.024,172.591,46.714,159.242
C08148=1030.530,370.240,-137.984,172.585,46.712,159.241
C08149=1030.521,369.993,-137.944,172.577,46.710,159.240
C08150=1030.513,369.746,-137.904,172.569,46.708,159.238
C08151=1030.505,369.500,-137.863,172.562,46.706,159.237
C08152=1030.496,369.253,-137.824,172.555,46.704,159.235
C08153=1030.488,369.006,-137.783,172.547,46.702,159.234
C08154=1030.479,368.760,-137.743,172.540,46.700,159.233
C08155=1030.471,368.513,-137.704,172.532,46.698,159.231
C08156=1030.463,368.267,-137.663,172.524,46.697,159.230
C08157=1030.454,368.020,-137.624,172.518,46.694,159.228
C08158=1030.445,367.773,-137.584,172.510,46.692,159.227
C08159=1030.438,367.526,-137.544,172.503,46.691,159.226
C08160=1030.429,367.280,-137.504,172.495,46.689,159.224
C08161=1030.420,367.034,-137.465,172.488,46.687,159.223
C08162=1030.413,366.787,-137.425,172.481,46.685,159.222
C08163=1030.404,366.540,-137.386,172.473,46.683,159.220
C08164=1030.396,366.293,-137.346,172.467,46.681,159.219
C08165=1030.388,366.047,-137.307,172.459,46.679,159.218
C08166=1030.380,365.800,-137.267,172.451,46.678,159.216
C08167=1030.373,365.587,-137.233,172.446,46.676,159.215
C08168=1030.365,365.375,-137.199,172.440,46.675,159.214
C08169=1030.359,365.163,-137.165,172.433,46.673,159.213
C08170=1030.351,364.951,-137.131,172.426,46.672,159.212
C08171=1030.345,364.740,-137.097,172.421,46.670,159.211
C08172=1030.337,364.527,-137.064,172.415,46.669,159.209
C08173=1030.330,364.316,-137.030,172.408,46.667,159.208
C08174=1030.323,364.103,-136.996,172.402,46.666,159.207
C08175=1030.315,363.857,-136.956,172.395,46.664,159.206
C08176=1030.307,363.610,-136.917,172.388,46.662,159.205
C08177=1030.298,363.363,-136.878,172.381,46.661,159.203
C08178=1030.290,363.116,-136.839,172.374,46.659,159.202
C08179=1030.283,362.870,-136.799,172.367,46.657,159.201
C08180=1030.274,362.623,-136.760,172.360,46.655,159.200
C08181=1030.266,362.376,-136.721,172.353,46.654,159.198
C08182=1030.259,362.129,-136.681,172.346,46.652,159.197
C08183=1030.250,361.883,-136.642,172.339,46.651,159.196
C08184=1030.242,361.635,-136.603,172.332,46.649,159.195
C08185=1030.235,361.389,-136.564,172.324,46.648,159.193
C08186=1030.227,361.142,-136.525,172.318,46.645,159.192
C08187=1030.218,360.895,-136.486,172.311,46.644,159.191
C08188=1030.210,360.648,-136.447,172.304,46.642,159.189
C08189=1030.202,360.402,-136.408,172.297,46.641,159.188
C08190=1030.194,360.155,-136.370,172.290,46.640,159.187
C08191=1030.186,359.908,-136.331,172.283,46.638,159.186
C08192=1030.177,359.661,-136.292,172.277,46.636,159.185
C08193=1030.169,359.414,-136.253,172.269,46.635,159.184
C08194=1030.162,359.168,-136.215,172.263,46.633,159.182
C08195=1030.154,358.920,-136.176,172.255,46.632,159.181
C08196=1030.145,358.674,-136.137,172.249,46.630,159.180
C08197=1030.138,358.427,-136.099,172.242,46.629,159.179
C08198=1030.129,358.180,-136.060,172.235,46.628,159.178
C08199=1030.121,357.933,-136.022,172.228,46.626,159.176
C08200=1030.114,357.686,-135.983,172.222,46.624,159.175
C08201=1030.106,357.439,-135.945,172.215,46.624,159.174
C08202=1030.097,357.192,-135.906,172.208,46.622,159.173
C08203=1030.090,356.945,-135.868,172.202,46.620,159.172
C08204=1030.082,356.698,-135.829,172.194,46.619,159.171
C08205=1030.074,356.452,-135.791,172.188,46.618,159.169
C08206=1030.066,356.204,-135.752,172.181,46.616,159.168
C08207=1030.058,355.957,-135.714,172.175,46.615,159.167
C08208=1030.050,355.711,-135.676,172.168,46.613,159.166
C08209=1030.042,355.463,-135.637,172.161,46.612,159.165
C08210=1030.035,355.217,-135.599,172.155,46.611,159.164
C08211=1030.026,354.970,-135.560,172.149,46.610,159.163
C08212=1030.019,354.723,-135.522,172.141,46.608,159.161
C08213=1030.010,354.476,-135.485,172.135,46.607,159.160
C08214=1030.003,354.229,-135.446,172.129,46.606,159.159
C08215=1029.995,353.982,-135.408,172.121,46.604,159.158
C08216=1029.987,353.735,-135.370,172.115,46.603,159.157
C08217=1029.979,353.488,-135.332,172.108,46.602,159.156
C08218=1029.971,353.241,-135.294,172.102,46.601,159.155
C08219=1029.963,352.994,-135.256,172.096,46.599,159.154
C08220=1029.956,352.747,-135.218,172.089,46.599,159.153
C08221=1029.947,352.501,-135.180,172.082,46.597,159.152
C08222=1029.939,352.253,-135.142,172.076,46.596,159.151
C08223=1029.932,352.006,-135.104,172.070,46.595,159.149
C08224=1029.925,351.759,-135.067,172.063,46.594,159.148
C08225=1029.916,351.512,-135.029,172.056,46.592,159.147
C08226=1029.909,351.265,-134.991,172.050,46.591,159.146
C08227=1029.895,350.848,-134.927,172.040,46.589,159.144
C08228=1029.883,350.430,-134.863,172.028,46.587,159.143
C08229=1029.869,350.012,-134.799,172.017,46.585,159.141
C08230=1029.857,349.594,-134.736,172.007,46.583,159.139
C08231=1029.848,349.347,-134.697,172.000,46.582,159.138
C08232=1029.840,349.100,-134.660,171.994,46.581,159.137
C08233=1029.833,348.853,-134.623,171.987,46.580,159.136
C08234=1029.826,348.606,-134.585,171.981,46.579,159.135
C08235=1029.817,348.358,-134.548,171.975,46.578,159.134
C08236=1029.810,348.111,-134.510,171.969,46.577,159.133
C08237=1029.802,347.864,-134.473,171.963,46.576,159.132
C08238=1029.795,347.618,-134.435,171.957,46.575,159.131
C08239=1029.787,347.371,-134.398,171.950,46.574,159.130
C08240=1029.779,347.123,-134.360,171.944,46.573,159.129
C08241=1029.771,346.876,-134.323,171.937,46.572,159.128
C08242=1029.764,346.629,-134.287,171.931,46.571,159.127
C08243=1029.756,346.382,-134.250,171.925,46.570,159.126
C08244=1029.749,346.135,-134.212,171.919,46.569,159.125
C08245=1029.741,345.888,-134.175,171.912,46.568,159.124
C08246=1029.733,345.641,-134.138,171.906,46.568,159.123
C08247=1029.725,345.394,-134.101,171.900,46.566,159.122
C08248=1029.718,345.147,-134.063,171.894,46.565,159.121
C08249=1029.710,344.899,-134.026,171.888,46.565,159.120
C08250=1029.703,344.652,-133.989,171.882,46.564,159.119
C08251=1029.695,344.405,-133.952,171.876,46.563,159.118
C08252=1029.687,344.158,-133.915,171.870,46.562,159.118
C08253=1029.679,343.911,-133.878,171.863,46.561,159.116
C08254=1029.673,343.663,-133.841,171.858,46.560,159.116
C08255=1029.665,343.416,-133.804,171.851,46.559,159.115
C08256=1029.657,343.169,-133.767,171.845,46.558,159.114
C08257=1029.650,342.922,-133.730,171.839,46.558,159.113
C08258=1029.642,342.675,-133.693,171.833,46.557,159.112
C08259=1029.635,342.427,-133.657,171.827,46.556,159.111
C08260=1029.627,342.180,-133.620,171.821,46.556,159.110
C08261=1029.619,341.934,-133.583,171.815,46.554,159.109
C08262=1029.612,341.686,-133.546,171.809,46.554,159.108
C08263=1029.604,341.440,-133.509,171.803,46.553,159.107
C08264=1029.597,341.192,-133.473,171.798,46.552,159.106
C08265=1029.590,340.944,-133.436,171.792,46.551,159.105
C08266=1029.582,340.697,-133.399,171.786,46.550,159.105
C08267=1029.575,340.450,-133.363,171.780,46.550,159.104
C08268=1029.567,340.203,-133.326,171.774,46.549,159.103
C08269=1029.559,339.955,-133.289,171.768,46.548,159.102
C08270=1029.552,339.709,-133.254,171.762,46.548,159.101
C08271=1029.544,339.461,-133.217,171.756,46.547,159.100
C08272=1029.536,339.214,-133.180,171.750,46.547,159.099
C08273=1029.529,338.967,-133.144,171.744,46.545,159.098
C08274=1029.522,338.719,-133.107,171.738,46.545,159.098
C08275=1029.514,338.472,-133.071,171.732,46.544,159.097
C08276=1029.507,338.225,-133.035,171.726,46.544,159.096
C08277=1029.499,337.978,-132.999,171.721,46.543,159.095
C08278=1029.491,337.731,-132.962,171.715,46.543,159.094
C08279=1029.484,337.483,-132.926,171.709,46.542,159.093
C08280=1029.477,337.237,-132.890,171.703,46.542,159.093
C08281=1029.470,336.989,-132.853,171.697,46.540,159.092
C08282=1029.462,336.741,-132.817,171.691,46.540,159.091
C08283=1029.456,336.531,-132.786,171.686,46.540,159.090
C08284=1029.449,336.320,-132.755,171.682,46.539,159.089
C08285=1029.443,336.110,-132.725,171.677,46.539,159.089
C08286=1029.437,335.900,-132.695,171.672,46.538,159.088
C08287=1029.431,335.689,-132.664,171.667,46.538,159.087
C08288=1029.424,335.479,-132.633,171.662,46.537,159.087
C08289=1029.418,335.268,-132.602,171.657,46.537,159.086
C08290=1029.412,335.057,-132.571,171.652,46.536,159.085
C08291=1029.405,334.811,-132.535,171.647,46.536,159.084
C08292=1029.397,334.563,-132.499,171.641,46.535,159.084
C08293=1029.390,334.315,-132.463,171.635,46.534,159.083
C08294=1029.383,334.068,-132.427,171.629,46.534,159.082
C08295=1029.375,333.821,-132.391,171.624,46.534,159.081
C08296=1029.368,333.574,-132.355,171.619,46.533,159.080
C08297=1029.360,333.326,-132.320,171.613,46.533,159.080
C08298=1029.353,333.079,-132.284,171.607,46.532,159.079
C08299=1029.345,332.832,-132.248,171.601,46.532,159.078
C08300=1029.338,332.584,-132.213,171.595,46.532,159.077
C08301=1029.331,332.338,-132.177,171.590,46.531,159.077
C08302=1029.323,332.089,-132.141,171.584,46.530,159.076
C08303=1029.316,331.843,-132.106,171.579,46.530,159.075
C08304=1029.308,331.595,-132.069,171.573,46.530,159.074
C08305=1029.301,331.347,-132.034,171.567,46.529,159.073
C08306=1029.293,331.101,-131.999,171.562,46.529,159.073
C08307=1029.286,330.853,-131.963,171.556,46.529,159.072
C08308=1029.279,330.606,-131.927,171.551,46.528,159.071
C08309=1029.272,330.359,-131.892,171.545,46.528,159.070
C08310=1029.264,330.111,-131.856,171.540,46.527,159.070
C08311=1029.258,329.864,-131.821,171.534,46.528,159.069
C08312=1029.250,329.616,-131.785,171.528,46.527,159.068
C08313=1029.242,329.369,-131.750,171.523,46.526,159.067
C08314=1029.235,329.121,-131.715,171.518,46.526,159.067
C08315=1029.228,328.874,-131.679,171.512,46.526,159.066
C08316=1029.221,328.627,-131.644,171.506,46.526,159.065
C08317=1029.214,328.379,-131.608,171.501,46.525,159.064
C08318=1029.207,328.132,-131.573,171.496,46.525,159.064
C08319=1029.199,327.884,-131.537,171.490,46.525,159.063
C08320=1029.192,327.637,-131.502,171.485,46.524,159.062
C08321=1029.185,327.390,-131.467,171.480,46.524,159.062
C08322=1029.177,327.142,-131.432,171.474,46.524,159.061
C08323=1029.170,326.895,-131.397,171.468,46.524,159.060
C08324=1029.162,326.647,-131.362,171.463,46.524,159.060
C08325=1029.155,326.400,-131.328,171.458,46.524,159.059
C08326=1029.148,326.153,-131.292,171.452,46.523,159.058
C08327=1029.140,325.905,-131.258,171.447,46.523,159.058
C08328=1029.133,325.657,-131.222,171.442,46.523,159.057
C08329=1029.125,325.410,-131.188,171.436,46.523,159.056
C08330=1029.118,325.162,-131.152,171.430,46.523,159.056
C08331=1029.111,324.915,-131.118,171.425,46.523,159.055
C08332=1029.103,324.668,-131.083,171.420,46.523,159.054
C08333=1029.096,324.420,-131.048,171.414,46.523,159.054
C08334=1029.088,324.173,-131.013,171.410,46.523,159.053
C08335=1029.082,323.925,-130.979,171.404,46.523,159.052
C08336=1029.074,323.678,-130.944,171.398,46.523,159.052
C08337=1029.066,323.430,-130.909,171.394,46.522,159.051
C08338=1029.059,323.183,-130.874,171.388,46.523,159.050
C08339=1029.052,322.936,-130.840,171.382,46.523,159.050
C08340=1029.045,322.688,-130.805,171.378,46.522,159.049
C08341=1029.038,322.441,-130.771,171.372,46.522,159.048
C08342=1029.030,322.193,-130.736,171.367,46.522,159.048
C08343=1029.024,321.980,-130.705,171.363,46.522,159.047
C08344=1029.018,321.767,-130.676,171.358,46.522,159.047
C08345=1029.011,321.555,-130.647,171.354,46.522,159.046
C08346=1029.006,321.342,-130.616,171.349,46.522,159.045
C08347=1028.999,321.129,-130.587,171.345,46.522,159.045
C08348=1028.993,320.917,-130.557,171.340,46.522,159.044
C08349=1028.987,320.704,-130.528,171.336,46.522,159.044
C08350=1028.981,320.491,-130.498,171.331,46.522,159.043
C08351=1028.974,320.244,-130.463,171.326,46.522,159.043
C08352=1028.966,319.996,-130.430,171.321,46.522,159.042
C08353=1028.960,319.749,-130.394,171.315,46.522,159.042
C08354=1028.952,319.501,-130.361,171.310,46.522,159.041
C08355=1028.946,319.254,-130.325,171.305,46.522,159.040
C08356=1028.938,319.007,-130.291,171.299,46.522,159.040
C08357=1028.931,318.759,-130.257,171.295,46.522,159.039
C08358=1028.924,318.511,-130.223,171.290,46.522,159.039
C08359=1028.917,318.264,-130.188,171.285,46.522,159.038
C08360=1028.910,318.016,-130.154,171.279,46.522,159.037
C08361=1028.903,317.769,-130.119,171.275,46.522,159.037
C08362=1028.896,317.521,-130.085,171.269,46.522,159.036
C08363=1028.889,317.274,-130.050,171.264,46.523,159.036
C08364=1028.882,317.026,-130.016,171.259,46.523,159.035
C08365=1028.875,316.778,-129.983,171.253,46.523,159.034
C08366=1028.868,316.531,-129.947,171.249,46.522,159.034
C08367=1028.861,316.283,-129.914,171.243,46.523,159.033
C08368=1028.853,316.036,-129.880,171.239,46.523,159.033
C08369=1028.847,315.788,-129.845,171.233,46.523,159.032
C08370=1028.840,315.541,-129.811,171.229,46.523,159.031
C08371=1028.833,315.294,-129.777,171.223,46.524,159.031
C08372=1028.826,315.046,-129.743,171.219,46.523,159.030
C08373=1028.819,314.799,-129.708,171.213,46.523,159.030
C08374=1028.812,314.551,-129.675,171.209,46.524,159.029
C08375=1028.805,314.303,-129.640,171.203,46.524,159.029
C08376=1028.798,314.055,-129.606,171.198,46.524,159.028
C08377=1028.791,313.808,-129.573,171.194,46.524,159.028
C08378=1028.785,313.561,-129.538,171.188,46.524,159.027
C08379=1028.778,313.313,-129.504,171.184,46.524,159.026
C08380=1028.771,313.065,-129.470,171.179,46.525,159.026
C08381=1028.764,312.818,-129.436,171.174,46.524,159.025
C08382=1028.757,312.571,-129.402,171.169,46.525,159.025
C08383=1028.751,312.323,-129.368,171.164,46.525,159.024
C08384=1028.744,312.075,-129.334,171.158,46.525,159.023
C08385=1028.736,311.827,-129.300,171.154,46.525,159.023
C08386=1028.730,311.580,-129.267,171.149,46.525,159.022
C08387=1028.723,311.332,-129.232,171.144,46.526,159.022
C08388=1028.716,311.085,-129.198,171.139,46.526,159.021
C08389=1028.710,310.838,-129.165,171.134,46.526,159.021
C08390=1028.702,310.590,-129.131,171.130,46.527,159.020
C08391=1028.695,310.342,-129.097,171.124,46.527,159.020
C08392=1028.687,310.094,-129.065,171.120,46.527,159.019
C08393=1028.681,309.847,-129.031,171.114,46.528,159.019
C08394=1028.674,309.600,-128.998,171.110,46.528,159.018
C08395=1028.667,309.351,-128.964,171.104,46.528,159.018
C08396=1028.659,309.104,-128.931,171.100,46.529,159.017
C08397=1028.652,308.857,-128.898,171.095,46.530,159.017
C08398=1028.645,308.609,-128.865,171.091,46.530,159.016
C08399=1028.637,308.362,-128.831,171.085,46.531,159.016
C08400=1028.631,308.113,-128.798,171.081,46.531,159.016
C08401=1028.624,307.866,-128.765,171.076,46.531,159.015
C08402=1028.617,307.619,-128.731,171.071,46.532,159.014
C08403=1028.610,307.408,-128.703,171.067,46.532,159.014
C08404=1028.605,307.198,-128.675,171.063,46.532,159.014
C08405=1028.599,306.988,-128.647,171.059,46.533,159.013
C08406=1028.592,306.778,-128.619,171.055,46.533,159.013
C08407=1028.586,306.567,-128.591,171.050,46.533,159.012
C08408=1028.581,306.357,-128.563,171.047,46.534,159.012
C08409=1028.575,306.146,-128.534,171.043,46.535,159.012
C08410=1028.569,305.937,-128.507,171.039,46.535,159.011
C08411=1028.562,305.689,-128.474,171.034,46.535,159.011
C08412=1028.555,305.442,-128.440,171.029,46.536,159.011
C08413=1028.548,305.194,-128.408,171.025,46.537,159.010
C08414=1028.540,304.946,-128.374,171.019,46.537,159.010
C08415=1028.534,304.698,-128.341,171.015,46.537,159.009
C08416=1028.527,304.450,-128.308,171.010,46.537,159.009
C08417=1028.520,304.203,-128.275,171.005,46.538,159.008
C08418=1028.513,303.955,-128.242,171.001,46.539,159.008
C08419=1028.507,303.707,-128.209,170.995,46.539,159.007
C08420=1028.499,303.460,-128.176,170.991,46.540,159.007
C08421=1028.492,303.213,-128.143,170.987,46.541,159.007
C08422=1028.486,302.964,-128.110,170.982,46.541,159.006
C08423=1028.479,302.717,-128.078,170.977,46.542,159.006
C08424=1028.471,302.469,-128.044,170.973,46.542,159.005
C08425=1028.465,302.222,-128.011,170.968,46.543,159.005
C08426=1028.457,301.974,-127.979,170.963,46.543,159.004
C08427=1028.451,301.726,-127.946,170.959,46.544,159.004
C08428=1028.444,301.478,-127.913,170.954,46.544,159.003
C08429=1028.437,301.231,-127.880,170.949,46.545,159.003
C08430=1028.430,300.983,-127.847,170.945,46.545,159.003
C08431=1028.424,300.735,-127.814,170.940,46.546,159.002
C08432=1028.417,300.488,-127.782,170.936,46.547,159.002
C08433=1028.410,300.240,-127.749,170.931,46.547,159.001
C08434=1028.404,299.992,-127.716,170.926,46.548,159.001
C08435=1028.397,299.744,-127.683,170.922,46.549,159.000
C08436=1028.390,299.496,-127.651,170.917,46.549,159.000
C08437=1028.383,299.249,-127.618,170.912,46.550,159.000
C08438=1028.376,299.001,-127.585,170.908,46.551,158.999
C08439=1028.369,298.753,-127.553,170.904,46.551,158.999
C08440=1028.363,298.506,-127.520,170.898,46.552,158.998
C08441=1028.356,298.257,-127.487,170.894,46.552,158.998
C08442=1028.349,298.010,-127.455,170.890,46.553,158.998
C08443=1028.343,297.763,-127.422,170.885,46.554,158.997
C08444=1028.336,297.514,-127.389,170.880,46.554,158.997
C08445=1028.329,297.267,-127.357,170.876,46.555,158.996
C08446=1028.323,297.019,-127.324,170.872,46.556,158.996
C08447=1028.316,296.772,-127.292,170.867,46.556,158.996
C08448=1028.309,296.524,-127.259,170.862,46.557,158.995
C08449=1028.302,296.276,-127.226,170.858,46.557,158.995
C08450=1028.296,296.028,-127.194,170.854,46.558,158.995
C08451=1028.289,295.781,-127.162,170.849,46.559,158.994
C08452=1028.283,295.532,-127.129,170.844,46.559,158.994
C08453=1028.276,295.285,-127.096,170.840,46.560,158.993
C08454=1028.269,295.038,-127.064,170.836,46.561,158.993
C08455=1028.263,294.789,-127.032,170.832,46.562,158.993
C08456=1028.257,294.542,-126.999,170.826,46.563,158.992
C08457=1028.249,294.294,-126.967,170.822,46.563,158.992
C08458=1028.243,294.046,-126.934,170.818,46.564,158.992
C08459=1028.236,293.798,-126.903,170.814,46.565,158.991
C08460=1028.229,293.551,-126.871,170.809,46.566,158.991
C08461=1028.223,293.302,-126.838,170.804,46.566,158.990
C08462=1028.216,293.055,-126.806,170.800,46.567,158.990
C08463=1028.204,292.652,-126.754,170.793,46.568,158.990
C08464=1028.194,292.249,-126.702,170.785,46.570,158.989
C08465=1028.182,291.845,-126.650,170.778,46.572,158.989
C08466=1028.172,291.441,-126.598,170.771,46.573,158.988
C08467=1028.165,291.194,-126.566,170.767,46.574,158.988
C08468=1028.158,290.946,-126.534,170.763,46.575,158.987
C08469=1028.151,290.698,-126.503,170.758,46.575,158.987
C08470=1028.144,290.450,-126.470,170.754,46.577,158.987
C08471=1028.137,290.202,-126.439,170.750,46.578,158.986
C08472=1028.131,289.954,-126.407,170.745,46.578,158.986
C08473=1028.124,289.707,-126.375,170.741,46.579,158.986
C08474=1028.117,289.459,-126.343,170.736,46.580,158.985
C08475=1028.111,289.211,-126.312,170.732,46.581,158.985
C08476=1028.104,288.964,-126.280,170.728,46.582,158.985
C08477=1028.098,288.716,-126.248,170.724,46.583,158.985
C08478=1028.091,288.468,-126.216,170.719,46.584,158.984
C08479=1028.084,288.220,-126.185,170.715,46.585,158.984
C08480=1028.076,287.972,-126.152,170.710,46.586,158.984
C08481=1028.070,287.724,-126.121,170.706,46.587,158.983
C08482=1028.063,287.476,-126.089,170.702,46.588,158.983
C08483=1028.056,287.228,-126.058,170.697,46.589,158.983
C08484=1028.050,286.980,-126.026,170.693,46.590,158.982
C08485=1028.044,286.732,-125.994,170.689,46.590,158.982
C08486=1028.037,286.484,-125.963,170.685,46.592,158.982
C08487=1028.030,286.236,-125.932,170.681,46.593,158.982
C08488=1028.023,285.989,-125.899,170.676,46.594,158.981
C08489=1028.016,285.741,-125.868,170.672,46.595,158.981
C08490=1028.010,285.493,-125.837,170.668,46.596,158.981
C08491=1028.003,285.245,-125.805,170.664,46.597,158.980
C08492=1027.996,284.997,-125.774,170.660,46.598,158.980
C08493=1027.989,284.749,-125.744,170.654,46.599,158.980
C08494=1027.982,284.501,-125.712,170.650,46.600,158.980
C08495=1027.976,284.253,-125.681,170.646,46.601,158.979
C08496=1027.969,284.005,-125.649,170.642,46.603,158.979
C08497=1027.962,283.757,-125.618,170.638,46.604,158.979
C08498=1027.955,283.509,-125.586,170.634,46.605,158.979
C08499=1027.949,283.262,-125.555,170.629,46.606,158.978
C08500=1027.942,283.014,-125.524,170.625,46.607,158.978
C08501=1027.935,282.766,-125.492,170.621,46.608,158.978
C08502=1027.928,282.518,-125.462,170.617,46.609,158.978
C08503=1027.921,282.270,-125.431,170.613,46.610,158.977
C08504=1027.915,282.022,-125.399,170.609,46.611,158.977
C08505=1027.908,281.774,-125.368,170.604,46.612,158.977
C08506=1027.902,281.526,-125.337,170.600,46.614,158.977
C08507=1027.895,281.278,-125.306,170.596,46.615,158.976
C08508=1027.889,281.030,-125.274,170.592,46.616,158.976
C08509=1027.882,280.782,-125.243,170.588,46.617,158.976
C08510=1027.875,280.534,-125.213,170.584,46.618,158.976
C08511=1027.868,280.286,-125.181,170.579,46.620,158.975
C08512=1027.861,280.038,-125.150,170.575,46.621,158.975
C08513=1027.855,279.790,-125.119,170.571,46.622,158.975
C08514=1027.849,279.543,-125.088,170.567,46.623,158.975
C08515=1027.842,279.295,-125.057,170.563,46.625,158.975
C08516=1027.836,279.046,-125.026,170.559,46.626,158.974
C08517=1027.829,278.798,-124.995,170.555,46.627,158.974
C08518=1027.821,278.551,-124.964,170.551,46.628,158.974
C08519=1027.812,278.159,-124.916,170.544,46.630,158.973
C08520=1027.801,277.768,-124.866,170.538,46.632,158.973
C08521=1027.791,277.377,-124.817,170.531,46.634,158.973
C08522=1027.780,276.986,-124.769,170.525,46.636,158.972
C08523=1027.773,276.738,-124.738,170.521,46.637,158.972
C08524=1027.767,276.490,-124.708,170.516,46.638,158.972
C08525=1027.760,276.242,-124.677,170.513,46.640,158.972
C08526=1027.753,275.994,-124.646,170.509,46.641,158.972
C08527=1027.747,275.745,-124.615,170.505,46.643,158.971
C08528=1027.740,275.498,-124.584,170.501,46.644,158.971
C08529=1027.734,275.250,-124.554,170.497,46.645,158.971
C08530=1027.727,275.002,-124.524,170.493,46.646,158.971
C08531=1027.720,274.754,-124.493,170.489,46.647,158.971
C08532=1027.713,274.505,-124.462,170.485,46.648,158.970
C08533=1027.707,274.258,-124.432,170.480,46.650,158.970
C08534=1027.700,274.009,-124.401,170.476,46.651,158.970
C08535=1027.693,273.762,-124.371,170.472,46.653,158.970
C08536=1027.687,273.514,-124.340,170.468,46.654,158.970
C08537=1027.681,273.265,-124.309,170.465,46.656,158.970
C08538=1027.674,273.017,-124.279,170.460,46.657,158.969
C08539=1027.667,272.770,-124.248,170.457,46.659,158.969
C08540=1027.660,272.522,-124.218,170.453,46.660,158.969
C08541=1027.654,272.273,-124.187,170.449,46.661,158.969
C08542=1027.647,272.026,-124.158,170.445,46.662,158.969
C08543=1027.641,271.777,-124.127,170.441,46.664,158.969
C08544=1027.634,271.529,-124.097,170.436,46.665,158.968
C08545=1027.628,271.282,-124.066,170.432,46.667,158.968
C08546=1027.620,271.034,-124.036,170.428,46.668,158.968
C08547=1027.614,270.785,-124.005,170.425,46.670,158.968
C08548=1027.607,270.538,-123.975,170.421,46.671,158.968
C08549=1027.601,270.289,-123.944,170.417,46.673,158.968
C08550=1027.594,270.041,-123.914,170.413,46.674,158.967
C08551=1027.588,269.793,-123.884,170.409,46.675,158.967
C08552=1027.581,269.545,-123.854,170.405,46.677,158.967
C08553=1027.574,269.297,-123.824,170.401,46.678,158.967
C08554=1027.568,269.049,-123.793,170.397,46.680,158.967
C08555=1027.561,268.801,-123.763,170.394,46.681,158.967
C08556=1027.554,268.553,-123.734,170.390,46.682,158.966
C08557=1027.548,268.305,-123.703,170.386,46.684,158.966
C08558=1027.541,268.056,-123.673,170.381,46.686,158.966
C08559=1027.535,267.808,-123.643,170.377,46.687,158.966
C08560=1027.528,267.560,-123.613,170.373,46.689,158.966
C08561=1027.521,267.312,-123.583,170.370,46.690,158.966
C08562=1027.515,267.064,-123.552,170.366,46.692,158.966
C08563=1027.508,266.816,-123.523,170.362,46.693,158.965
C08564=1027.501,266.568,-123.493,170.358,46.695,158.965
C08565=1027.495,266.320,-123.462,170.354,46.697,158.965
C08566=1027.489,266.071,-123.433,170.351,46.698,158.965
C08567=1027.481,265.823,-123.403,170.347,46.699,158.965
C08568=1027.475,265.576,-123.373,170.343,46.701,158.965
C08569=1027.468,265.327,-123.343,170.339,46.703,158.965
C08570=1027.462,265.079,-123.313,170.335,46.704,158.965
C08571=1027.455,264.831,-123.283,170.332,46.706,158.965
C08572=1027.449,264.583,-123.253,170.328,46.708,158.965
C08573=1027.442,264.334,-123.224,170.324,46.709,158.964
C08574=1027.435,264.087,-123.194,170.320,46.711,158.964
C08575=1027.425,263.701,-123.148,170.314,46.714,158.964
C08576=1027.414,263.314,-123.101,170.308,46.716,158.964
C08577=1027.404,262.927,-123.055,170.302,46.718,158.964
C08578=1027.394,262.541,-123.009,170.297,46.721,158.964
C08579=1027.388,262.293,-122.979,170.293,46.723,158.964
C08580=1027.381,262.044,-122.949,170.289,46.724,158.963
C08581=1027.375,261.797,-122.919,170.285,46.725,158.963
C08582=1027.368,261.548,-122.890,170.281,46.727,158.963
C08583=1027.361,261.300,-122.860,170.278,46.729,158.963
C08584=1027.355,261.051,-122.830,170.274,46.730,158.963
C08585=1027.349,260.804,-122.800,170.270,46.732,158.963
C08586=1027.342,260.556,-122.772,170.265,46.734,158.963
C08587=1027.335,260.307,-122.742,170.262,46.736,158.963
C08588=1027.328,260.059,-122.713,170.258,46.738,158.963
C08589=1027.322,259.811,-122.683,170.254,46.740,158.963
C08590=1027.315,259.563,-122.654,170.251,46.742,158.963
C08591=1027.307,259.314,-122.625,170.247,46.743,158.962
C08592=1027.301,259.066,-122.596,170.243,46.745,158.962
C08593=1027.294,258.818,-122.566,170.239,46.747,158.962
C08594=1027.288,258.570,-122.537,170.236,46.748,158.962
C08595=1027.281,258.322,-122.508,170.232,46.751,158.962
C08596=1027.274,258.073,-122.479,170.228,46.752,158.962
C08597=1027.268,257.825,-122.450,170.225,46.754,158.962
C08598=1027.260,257.577,-122.420,170.221,46.756,158.962
C08599=1027.254,257.329,-122.391,170.217,46.757,158.962
C08600=1027.247,257.081,-122.362,170.214,46.760,158.962
C08601=1027.240,256.832,-122.333,170.210,46.761,158.962
C08602=1027.234,256.584,-122.304,170.206,46.763,158.962
C08603=1027.228,256.336,-122.275,170.202,46.765,158.962
C08604=1027.220,256.088,-122.245,170.199,46.767,158.962
C08605=1027.214,255.840,-122.216,170.195,46.769,158.962
C08606=1027.207,255.592,-122.187,170.192,46.771,158.962
C08607=1027.201,255.343,-122.158,170.188,46.772,158.962
C08608=1027.194,255.095,-122.129,170.184,46.774,158.962
C08609=1027.187,254.847,-122.100,170.181,46.776,158.962
C08610=1027.181,254.598,-122.071,170.177,46.778,158.962
C08611=1027.174,254.350,-122.042,170.173,46.780,158.961
C08612=1027.168,254.102,-122.013,170.170,46.782,158.962
C08613=1027.160,253.853,-121.984,170.166,46.784,158.961
C08614=1027.154,253.605,-121.955,170.162,46.785,158.961
C08615=1027.148,253.357,-121.926,170.158,46.787,158.961
C08616=1027.142,253.109,-121.897,170.155,46.790,158.961
C08617=1027.134,252.860,-121.868,170.151,46.791,158.961
C08618=1027.128,252.612,-121.839,170.147,46.793,158.961
C08619=1027.122,252.364,-121.810,170.144,46.795,158.961
C08620=1027.115,252.116,-121.781,170.140,46.797,158.961
C08621=1027.108,251.868,-121.752,170.136,46.799,158.961
C08622=1027.102,251.619,-121.723,170.133,46.801,158.961
C08623=1027.095,251.371,-121.694,170.129,46.803,158.961
C08624=1027.089,251.123,-121.665,170.126,46.804,158.961
C08625=1027.082,250.875,-121.636,170.122,46.807,158.961
C08626=1027.075,250.627,-121.607,170.118,46.808,158.961
C08627=1027.069,250.378,-121.578,170.115,46.810,158.961
C08628=1027.063,250.130,-121.549,170.111,46.812,158.961
C08629=1027.056,249.882,-121.521,170.107,46.814,158.961
C08630=1027.050,249.634,-121.492,170.104,46.817,158.961
C08631=1027.040,249.246,-121.447,170.098,46.819,158.961
C08632=1027.029,248.857,-121.402,170.093,46.822,158.961
C08633=1027.020,248.470,-121.357,170.088,46.825,158.961
C08634=1027.009,248.082,-121.312,170.082,46.828,158.961
C08635=1027.003,247.834,-121.283,170.079,46.830,158.961
C08636=1026.996,247.586,-121.254,170.075,46.832,158.961
C08637=1026.990,247.337,-121.225,170.071,46.834,158.961
C08638=1026.983,247.089,-121.197,170.068,46.836,158.961
C08639=1026.977,246.840,-121.168,170.064,46.838,158.961
C08640=1026.970,246.592,-121.139,170.060,46.840,158.961
C08641=1026.964,246.344,-121.110,170.057,46.842,158.961
C08642=1026.957,246.096,-121.082,170.053,46.844,158.961
C08643=1026.951,245.848,-121.053,170.049,46.846,158.961
C08644=1026.945,245.599,-121.024,170.046,46.848,158.961
C08645=1026.939,245.351,-120.995,170.042,46.850,158.961
C08646=1026.932,245.103,-120.967,170.040,46.852,158.961
C08647=1026.926,244.854,-120.939,170.036,46.854,158.961
C08648=1026.920,244.606,-120.910,170.033,46.856,158.961
C08649=1026.913,244.358,-120.881,170.029,46.858,158.961
C08650=1026.907,244.109,-120.853,170.025,46.860,158.961
C08651=1026.901,243.861,-120.824,170.022,46.862,158.961
C08652=1026.894,243.613,-120.796,170.018,46.864,158.961
C08653=1026.888,243.365,-120.767,170.015,46.867,158.961
C08654=1026.881,243.116,-120.739,170.011,46.868,158.961
C08655=1026.874,242.868,-120.711,170.008,46.871,158.961
C08656=1026.868,242.620,-120.682,170.004,46.873,158.961
C08657=1026.861,242.372,-120.654,170.000,46.875,158.961
C08658=1026.855,242.122,-120.625,169.998,46.877,158.961
C08659=1026.848,241.875,-120.597,169.995,46.879,158.961
C08660=1026.842,241.626,-120.569,169.991,46.881,158.961
C08661=1026.835,241.377,-120.541,169.987,46.883,158.961
C08662=1026.829,241.129,-120.512,169.984,46.886,158.961
C08663=1026.822,240.881,-120.484,169.980,46.887,158.961
C08664=1026.816,240.633,-120.455,169.977,46.890,158.961
C08665=1026.810,240.385,-120.428,169.973,46.892,158.961
C08666=1026.803,240.137,-120.400,169.970,46.894,158.961
C08667=1026.797,239.888,-120.371,169.966,46.896,158.961
C08668=1026.790,239.640,-120.343,169.963,46.898,158.961
C08669=1026.783,239.391,-120.315,169.959,46.901,158.961
C08670=1026.777,239.143,-120.288,169.956,46.903,158.962
C08671=1026.770,238.895,-120.259,169.953,46.905,158.962
C08672=1026.764,238.646,-120.231,169.950,46.907,158.962
C08673=1026.757,238.398,-120.203,169.946,46.909,158.962
C08674=1026.750,238.150,-120.175,169.943,46.912,158.962
C08675=1026.744,237.901,-120.148,169.939,46.914,158.962
C08676=1026.738,237.653,-120.119,169.936,46.916,158.962
C08677=1026.731,237.405,-120.091,169.932,46.919,158.962
C08678=1026.724,237.156,-120.063,169.929,46.921,158.962
C08679=1026.717,236.908,-120.035,169.925,46.923,158.962
C08680=1026.711,236.659,-120.008,169.922,46.925,158.962
C08681=1026.705,236.410,-119.979,169.918,46.927,158.962
C08682=1026.698,236.162,-119.952,169.915,46.930,158.962
C08683=1026.691,235.914,-119.924,169.911,46.932,158.962
C08684=1026.684,235.666,-119.896,169.908,46.935,158.962
C08685=1026.678,235.418,-119.868,169.905,46.937,158.963
C08686=1026.672,235.170,-119.840,169.902,46.939,158.963
C08687=1026.661,234.775,-119.797,169.896,46.943,158.963
C08688=1026.651,234.381,-119.752,169.891,46.946,158.963
C08689=1026.641,233.987,-119.708,169.886,46.951,158.963
C08690=1026.630,233.592,-119.664,169.881,46.954,158.963
C08691=1026.624,233.344,-119.637,169.877,46.956,158.963
C08692=1026.617,233.096,-119.609,169.874,46.959,158.963
C08693=1026.611,232.848,-119.582,169.870,46.961,158.963
C08694=1026.605,232.599,-119.553,169.867,46.964,158.963
C08695=1026.598,232.351,-119.526,169.863,46.966,158.964
C08696=1026.591,232.102,-119.498,169.860,46.968,158.964
C08697=1026.585,231.854,-119.470,169.857,46.970,158.964
C08698=1026.578,231.605,-119.442,169.854,46.973,158.964
C08699=1026.572,231.358,-119.415,169.851,46.975,158.964
C08700=1026.565,231.109,-119.387,169.847,46.977,158.964
C08701=1026.559,230.860,-119.360,169.844,46.980,158.964
C08702=1026.552,230.612,-119.333,169.840,46.982,158.964
C08703=1026.546,230.363,-119.305,169.837,46.985,158.964
C08704=1026.540,230.115,-119.277,169.833,46.987,158.964
C08705=1026.533,229.867,-119.250,169.830,46.989,158.964
C08706=1026.526,229.618,-119.223,169.826,46.992,158.965
C08707=1026.520,229.369,-119.195,169.824,46.994,158.965
C08708=1026.514,229.122,-119.168,169.821,46.997,158.965
C08709=1026.507,228.873,-119.140,169.817,46.999,158.965
C08710=1026.501,228.624,-119.113,169.814,47.001,158.965
C08711=1026.494,228.376,-119.085,169.810,47.004,158.965
C08712=1026.487,228.127,-119.057,169.807,47.006,158.965
C08713=1026.481,227.880,-119.030,169.804,47.009,158.965
C08714=1026.475,227.631,-119.003,169.800,47.012,158.966
C08715=1026.468,227.382,-118.975,169.797,47.014,158.966
C08716=1026.461,227.135,-118.949,169.795,47.016,158.966
C08717=1026.455,226.886,-118.921,169.791,47.018,158.966
C08718=1026.448,226.637,-118.894,169.788,47.021,158.966
C08719=1026.442,226.388,-118.867,169.784,47.024,158.966
C08720=1026.435,226.141,-118.840,169.781,47.026,158.966
C08721=1026.429,225.892,-118.813,169.778,47.029,158.967
C08722=1026.422,225.643,-118.785,169.774,47.032,158.967
C08723=1026.415,225.395,-118.758,169.771,47.034,158.967
C08724=1026.409,225.147,-118.731,169.768,47.037,158.967
C08725=1026.402,224.898,-118.704,169.764,47.039,158.967
C08726=1026.396,224.649,-118.677,169.761,47.042,158.967
C08727=1026.388,224.401,-118.650,169.759,47.044,158.967
C08728=1026.383,224.153,-118.623,169.755,47.047,158.967
C08729=1026.376,223.904,-118.595,169.752,47.049,158.968
C08730=1026.369,223.655,-118.569,169.749,47.052,158.968
C08731=1026.363,223.407,-118.542,169.745,47.055,158.968
C08732=1026.356,223.159,-118.514,169.742,47.057,158.968
C08733=1026.350,222.910,-118.487,169.739,47.060,158.968
C08734=1026.343,222.662,-118.461,169.735,47.062,158.968
C08735=1026.337,222.413,-118.434,169.732,47.065,158.969
C08736=1026.330,222.165,-118.406,169.730,47.067,158.969
C08737=1026.324,221.917,-118.380,169.726,47.070,158.969
C08738=1026.317,221.668,-118.353,169.723,47.073,158.969
C08739=1026.311,221.419,-118.325,169.720,47.075,158.969
C08740=1026.305,221.171,-118.298,169.716,47.078,158.969
C08741=1026.297,220.923,-118.271,169.713,47.081,158.969
C08742=1026.292,220.674,-118.245,169.710,47.083,158.969
C08743=1026.281,220.272,-118.201,169.705,47.087,158.970
C08744=1026.270,219.870,-118.158,169.700,47.091,158.970
C08745=1026.260,219.469,-118.114,169.694,47.096,158.970
C08746=1026.250,219.067,-118.070,169.689,47.100,158.971
C08747=1026.243,218.818,-118.043,169.686,47.103,158.971
C08748=1026.236,218.569,-118.017,169.683,47.106,158.971
C08749=1026.230,218.321,-117.990,169.680,47.108,158.971
C08750=1026.223,218.073,-117.963,169.677,47.111,158.971
C08751=1026.216,217.825,-117.937,169.674,47.114,158.972
C08752=1026.210,217.576,-117.910,169.670,47.116,158.972
C08753=1026.203,217.328,-117.884,169.667,47.119,158.972
C08754=1026.197,217.079,-117.857,169.664,47.122,158.972
C08755=1026.190,216.830,-117.831,169.661,47.125,158.972
C08756=1026.183,216.582,-117.805,169.658,47.128,158.972
C08757=1026.177,216.333,-117.778,169.654,47.130,158.972
C08758=1026.170,216.085,-117.751,169.651,47.133,158.973
C08759=1026.164,215.836,-117.724,169.649,47.136,158.973
C08760=1026.157,215.588,-117.698,169.645,47.138,158.973
C08761=1026.150,215.339,-117.671,169.642,47.141,158.973
C08762=1026.144,215.090,-117.644,169.639,47.144,158.974
C08763=1026.137,214.842,-117.618,169.636,47.147,158.974
C08764=1026.131,214.593,-117.591,169.633,47.150,158.974
C08765=1026.124,214.345,-117.565,169.629,47.153,158.974
C08766=1026.118,214.096,-117.538,169.626,47.155,158.974
C08767=1026.112,213.848,-117.512,169.623,47.158,158.975
C08768=1026.104,213.599,-117.486,169.621,47.161,158.975
C08769=1026.099,213.351,-117.459,169.617,47.163,158.975
C08770=1026.092,213.102,-117.433,169.614,47.166,158.975
C08771=1026.086,212.854,-117.406,169.611,47.169,158.975
C08772=1026.079,212.605,-117.380,169.608,47.172,158.975
C08773=1026.072,212.357,-117.354,169.604,47.175,158.976
C08774=1026.066,212.109,-117.327,169.601,47.178,158.976
C08775=1026.059,211.860,-117.300,169.599,47.180,158.976
C08776=1026.054,211.612,-117.274,169.596,47.183,158.976
C08777=1026.046,211.363,-117.247,169.593,47.186,158.977
C08778=1026.040,211.115,-117.221,169.589,47.189,158.977
C08779=1026.034,210.865,-117.195,169.586,47.191,158.977
C08780=1026.027,210.617,-117.169,169.583,47.194,158.977
C08781=1026.020,210.368,-117.143,169.580,47.197,158.977
C08782=1026.014,210.120,-117.116,169.578,47.200,158.978
C08783=1026.008,209.872,-117.090,169.574,47.203,158.978
C08784=1026.001,209.623,-117.063,169.571,47.206,158.978
C08785=1025.994,209.375,-117.037,169.568,47.209,158.978
C08786=1025.987,209.126,-117.012,169.565,47.212,158.979
C08787=1025.982,208.877,-116.985,169.562,47.215,158.979
C08788=1025.975,208.629,-116.959,169.558,47.218,158.979
C08789=1025.968,208.381,-116.933,169.555,47.220,158.979
C08790=1025.962,208.132,-116.907,169.552,47.223,158.979
C08791=1025.955,207.883,-116.881,169.550,47.226,158.980
C08792=1025.949,207.635,-116.854,169.547,47.229,158.980
C08793=1025.942,207.386,-116.828,169.544,47.232,158.980
C08794=1025.936,207.137,-116.802,169.540,47.235,158.980
C08795=1025.929,206.889,-116.776,169.537,47.238,158.981
C08796=1025.922,206.641,-116.750,169.534,47.241,158.981
C08797=1025.916,206.392,-116.725,169.531,47.244,158.981
C08798=1025.909,206.143,-116.698,169.528,47.247,158.981
C08799=1025.898,205.745,-116.657,169.523,47.252,158.982
C08800=1025.888,205.346,-116.615,169.518,47.257,158.982
C08801=1025.877,204.948,-116.574,169.514,47.261,158.983
C08802=1025.867,204.549,-116.532,169.508,47.267,158.983
C08803=1025.842,203.513,-116.430,169.115,47.165,158.911
C08804=1025.837,203.265,-116.406,169.111,47.168,158.911
C08805=1025.831,203.015,-116.381,169.107,47.172,158.912
C08806=1025.825,202.767,-116.357,169.103,47.176,158.912
C08807=1025.819,202.518,-116.333,169.098,47.179,158.912
C08808=1025.814,202.270,-116.308,169.094,47.183,158.912
C08809=1025.808,202.020,-116.283,169.090,47.187,158.913
C08810=1025.802,201.772,-116.260,169.086,47.191,158.913
C08811=1025.796,201.524,-116.235,169.082,47.195,158.913
C08812=1025.791,201.274,-116.211,169.078,47.199,158.914
C08813=1025.785,201.026,-116.186,169.074,47.203,158.914
C08814=1025.779,200.776,-116.162,169.071,47.207,158.914
C08815=1025.773,200.528,-116.138,169.066,47.210,158.914
C08816=1025.767,200.279,-116.113,169.063,47.214,158.915
C08817=1025.762,200.030,-116.089,169.059,47.218,158.915
C08818=1025.756,199.782,-116.066,169.055,47.222,158.915
C08819=1025.750,199.533,-116.041,169.051,47.226,158.916
C08820=1025.744,199.284,-116.017,169.047,47.230,158.916
C08821=1025.738,199.035,-115.993,169.043,47.234,158.916
C08822=1025.732,198.787,-115.969,169.039,47.238,158.917
C08823=1025.727,198.538,-115.945,169.036,47.242,158.917
C08824=1025.720,198.289,-115.921,169.032,47.246,158.917
C08825=1025.714,198.041,-115.897,169.028,47.250,158.918
C08826=1025.709,197.791,-115.873,169.024,47.254,158.918
C08827=1025.703,197.543,-115.849,169.020,47.258,158.918
C08828=1025.697,197.294,-115.825,169.015,47.261,158.918
C08829=1025.691,197.045,-115.801,169.011,47.265,158.919
C08830=1025.685,196.797,-115.777,169.007,47.269,158.919
C08831=1025.680,196.548,-115.754,169.003,47.273,158.919
C08832=1025.673,196.299,-115.730,168.999,47.277,158.920
C08833=1025.668,196.050,-115.706,168.996,47.281,158.920
C08834=1025.662,195.802,-115.682,168.992,47.285,158.920
C08835=1025.656,195.552,-115.658,168.988,47.289,158.921
C08836=1025.650,195.304,-115.634,168.984,47.293,158.921
C08837=1025.644,195.055,-115.611,168.980,47.297,158.921
C08838=1025.638,194.806,-115.586,168.976,47.301,158.922
C08839=1025.632,194.557,-115.563,168.972,47.305,158.922
C08840=1025.627,194.309,-115.539,168.968,47.309,158.922
C08841=1025.620,194.060,-115.515,168.965,47.313,158.923
C08842=1025.615,193.810,-115.491,168.961,47.317,158.923
C08843=1025.609,193.562,-115.468,168.957,47.321,158.923
C08844=1025.603,193.314,-115.444,168.953,47.325,158.924
C08845=1025.598,193.064,-115.420,168.949,47.329,158.924
C08846=1025.592,192.816,-115.397,168.946,47.333,158.924
C08847=1025.587,192.567,-115.373,168.943,47.338,158.925
C08848=1025.581,192.318,-115.349,168.939,47.342,158.925
C08849=1025.575,192.070,-115.326,168.935,47.346,158.925
C08850=1025.569,191.820,-115.302,168.931,47.350,158.926
C08851=1025.563,191.572,-115.278,168.927,47.354,158.926
C08852=1025.558,191.323,-115.255,168.923,47.358,158.926
C08853=1025.552,191.074,-115.231,168.920,47.362,158.927
C08854=1025.546,190.825,-115.208,168.916,47.366,158.927
C08855=1025.540,190.576,-115.183,168.912,47.370,158.927
C08856=1025.535,190.327,-115.160,168.908,47.374,158.928
C08857=1025.529,190.079,-115.137,168.904,47.378,158.928
C08858=1025.524,189.830,-115.113,168.900,47.382,158.928
C08859=1025.518,189.581,-115.090,168.896,47.386,158.929
C08860=1025.513,189.332,-115.066,168.894,47.389,158.929
C08861=1025.506,189.083,-115.042,168.890,47.393,158.929
C08862=1025.500,188.834,-115.019,168.886,47.397,158.930
C08863=1025.495,188.586,-114.995,168.882,47.401,158.930
C08864=1025.488,188.303,-114.968,168.877,47.406,158.930
C08865=1025.483,188.021,-114.942,168.874,47.410,158.931
C08866=1025.476,187.738,-114.915,168.869,47.415,158.931
C08867=1025.469,187.456,-114.888,168.866,47.420,158.932
C08868=1025.464,187.206,-114.865,168.862,47.424,158.932
C08869=1025.458,186.958,-114.841,168.858,47.428,158.932
C08870=1025.452,186.709,-114.818,168.854,47.432,158.933
C08871=1025.447,186.460,-114.795,168.850,47.436,158.933
C08872=1025.441,186.212,-114.771,168.847,47.440,158.933
C08873=1025.435,185.963,-114.748,168.843,47.444,158.934
C08874=1025.430,185.714,-114.724,168.840,47.448,158.934
C08875=1025.424,185.465,-114.701,168.836,47.452,158.934
C08876=1025.419,185.216,-114.677,168.832,47.456,158.935
C08877=1025.414,184.967,-114.654,168.828,47.460,158.935
C08878=1025.407,184.718,-114.630,168.825,47.464,158.935
C08879=1025.402,184.469,-114.607,168.822,47.468,158.936
C08880=1025.396,184.220,-114.584,168.818,47.472,158.936
C08881=1025.390,183.972,-114.560,168.814,47.476,158.936
C08882=1025.385,183.723,-114.537,168.810,47.480,158.937
C08883=1025.380,183.474,-114.514,168.807,47.484,158.937
C08884=1025.374,183.225,-114.491,168.803,47.488,158.937
C08885=1025.369,182.976,-114.467,168.800,47.492,158.938
C08886=1025.363,182.727,-114.443,168.796,47.496,158.938
C08887=1025.358,182.478,-114.420,168.792,47.500,158.938
C08888=1025.351,182.230,-114.398,168.789,47.505,158.939
C08889=1025.346,181.981,-114.375,168.785,47.509,158.939
C08890=1025.340,181.732,-114.352,168.782,47.513,158.940
C08891=1025.334,181.483,-114.329,168.778,47.518,158.940
C08892=1025.328,181.234,-114.307,168.774,47.522,158.940
C08893=1025.322,180.985,-114.284,168.771,47.526,158.941
C08894=1025.317,180.736,-114.261,168.767,47.530,158.941
C08895=1025.311,180.487,-114.238,168.763,47.535,158.942
C08896=1025.304,180.238,-114.216,168.759,47.539,158.942
C08897=1025.299,179.990,-114.193,168.757,47.543,158.943
C08898=1025.293,179.741,-114.170,168.753,47.547,158.943
C08899=1025.287,179.492,-114.147,168.749,47.551,158.943
C08900=1025.281,179.243,-114.125,168.746,47.556,158.944
C08901=1025.275,178.994,-114.103,168.742,47.560,158.944
C08902=1025.270,178.745,-114.080,168.738,47.565,158.944
C08903=1025.263,178.496,-114.057,168.734,47.569,158.945
C08904=1025.257,178.247,-114.034,168.731,47.574,158.945
C08905=1025.252,177.998,-114.011,168.728,47.577,158.946
C08906=1025.246,177.749,-113.988,168.724,47.581,158.946
C08907=1025.240,177.500,-113.967,168.721,47.586,158.946
C08908=1025.234,177.251,-113.944,168.717,47.590,158.947
C08909=1025.228,177.002,-113.921,168.713,47.595,158.947
C08910=1025.223,176.754,-113.898,168.709,47.599,158.948
C08911=1025.216,176.504,-113.876,168.707,47.603,158.948
C08912=1025.211,176.255,-113.853,168.703,47.607,158.948
C08913=1025.205,176.007,-113.830,168.700,47.612,158.949
C08914=1025.200,175.758,-113.808,168.696,47.616,158.949
C08915=1025.194,175.509,-113.786,168.692,47.620,158.950
C08916=1025.188,175.260,-113.763,168.689,47.625,158.950
C08917=1025.182,175.011,-113.740,168.686,47.629,158.950
C08918=1025.176,174.762,-113.719,168.682,47.633,158.951
C08919=1025.170,174.513,-113.696,168.678,47.638,158.951
C08920=1025.165,174.264,-113.673,168.675,47.642,158.952
C08921=1025.159,174.015,-113.651,168.672,47.646,158.952
C08922=1025.153,173.767,-113.629,168.668,47.651,158.953
C08923=1025.147,173.518,-113.606,168.664,47.655,158.953
C08924=1025.142,173.269,-113.583,168.661,47.659,158.953
C08925=1025.136,173.020,-113.561,168.658,47.663,158.954
C08926=1025.130,172.771,-113.538,168.654,47.667,158.954
C08927=1025.124,172.522,-113.516,168.651,47.672,158.955
C08928=1025.118,172.239,-113.490,168.647,47.677,158.955
C08929=1025.111,171.956,-113.465,168.643,47.682,158.955
C08930=1025.105,171.673,-113.439,168.639,47.686,158.956
C08931=1025.099,171.390,-113.414,168.636,47.691,158.956
C08932=1025.093,171.141,-113.392,168.632,47.696,158.957
C08933=1025.087,170.892,-113.369,168.628,47.700,158.957
C08934=1025.082,170.643,-113.347,168.624,47.704,158.957
C08935=1025.076,170.394,-113.324,168.622,47.708,158.958
C08936=1025.070,170.145,-113.303,168.618,47.713,158.958
C08937=1025.064,169.896,-113.280,168.615,47.717,158.959
C08938=1025.059,169.647,-113.258,168.612,47.721,158.959
C08939=1025.053,169.399,-113.236,168.608,47.726,158.960
C08940=1025.048,169.149,-113.213,168.604,47.730,158.960
C08941=1025.042,168.900,-113.190,168.601,47.735,158.960
C08942=1025.037,168.651,-113.168,168.598,47.738,158.961
C08943=1025.031,168.403,-113.146,168.595,47.743,158.961
C08944=1025.025,168.154,-113.124,168.591,47.747,158.962
C08945=1025.020,167.905,-113.101,168.588,47.752,158.962
C08946=1025.013,167.655,-113.079,168.584,47.756,158.963
C08947=1025.008,167.407,-113.057,168.581,47.760,158.963
C08948=1025.003,167.158,-113.035,168.578,47.764,158.963
C08949=1024.997,166.909,-113.013,168.574,47.768,158.964
C08950=1024.992,166.660,-112.990,168.571,47.773,158.964
C08951=1024.986,166.411,-112.968,168.568,47.777,158.965
C08952=1024.980,166.162,-112.946,168.564,47.782,158.965
C08953=1024.975,165.913,-112.924,168.560,47.786,158.965
C08954=1024.969,165.664,-112.902,168.558,47.790,158.966
C08955=1024.964,165.415,-112.879,168.554,47.794,158.966
C08956=1024.958,165.167,-112.857,168.551,47.799,158.967
C08957=1024.953,164.917,-112.835,168.548,47.803,158.967
C08958=1024.947,164.668,-112.812,168.544,47.807,158.968
C08959=1024.941,164.420,-112.791,168.541,47.811,158.968
C08960=1024.936,164.170,-112.769,168.538,47.815,158.968
C08961=1024.931,163.922,-112.746,168.534,47.820,158.969
C08962=1024.925,163.673,-112.725,168.531,47.824,158.969
C08963=1024.919,163.423,-112.702,168.528,47.829,158.970
C08964=1024.914,163.175,-112.680,168.525,47.832,158.970
C08965=1024.908,162.926,-112.658,168.522,47.837,158.970
C08966=1024.903,162.677,-112.636,168.518,47.841,158.971
C08967=1024.898,162.427,-112.614,168.515,47.846,158.971
C08968=1024.891,162.179,-112.592,168.511,47.850,158.972
C08969=1024.886,161.930,-112.570,168.509,47.854,158.972
C08970=1024.881,161.681,-112.548,168.505,47.858,158.972
C08971=1024.875,161.432,-112.526,168.502,47.863,158.973
C08972=1024.870,161.183,-112.503,168.499,47.867,158.973
C08973=1024.865,160.934,-112.481,168.495,47.871,158.974
